KUKA KRL program: MyProgram_132().src

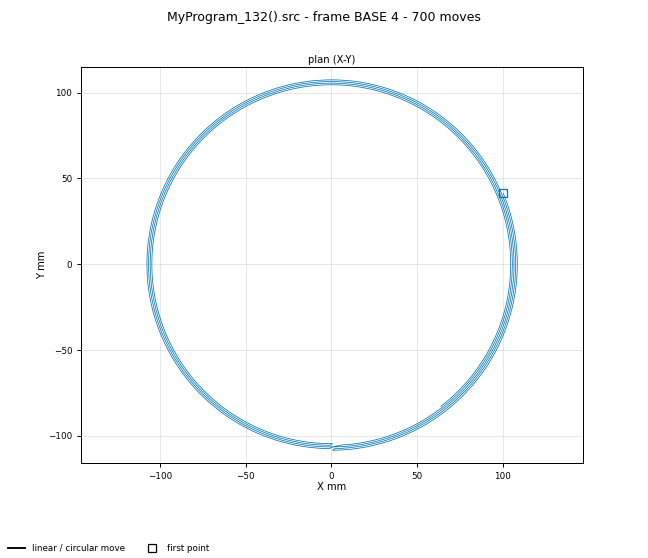
[picture p0: tool path of MyProgram_132().src in frame BASE 4, 700 of 700 moves have a stored position in this frame; points joined in program order, loops and branches not executed]
&ACCESS RVP
&REL 1
&PARAM TEMPLATE = C:\KRC\Roboter\Template\vorgabe
&PARAM EDITMASK = *
DEF MyProgram_132()
; ---- Setting reference (Base) ----
$BASE = BASE_DATA[4]

; --------------------------
; ---- Setting tool (TCP) ----
$TOOL = TOOL_DATA[3]
; --------------------------

$VEL.CP = VEL_APROX_PRINT
Startdeposition()
$VEL.CP = VEL_PRINT
LIN {X 100.2174,Y 41.413,Z 108,A 17.7358,B 24.9349,C -1.8633,E1 25.148,E2 427.9608} C_DIS
LIN {X 101.3618,Y 38.5229,Z 108,A 15.9205,B 24.9358,C -1.851,E1 25.1499,E2 429.795} C_DIS
LIN {X 102.6598,Y 34.9179,Z 108,A 13.9537,B 24.936,C -1.8475,E1 25.1517,E2 431.7591} C_DIS
LIN {X 103.7872,Y 31.4133,Z 108,A 11.2694,B 24.9386,C -1.8096,E1 25.154,E2 434.5174} C_DIS
LIN {X 105.0738,Y 26.7911,Z 108,A 10.0153,B 24.9353,C -1.8575,E1 25.1548,E2 435.6515} C_DIS
LIN {X 105.9493,Y 23.0863,Z 108,A 7.5492,B 24.9371,C -1.8313,E1 25.1564,E2 438.165} C_DIS
LIN {X 107.0471,Y 17.303,Z 108,A 4.2698,B 24.9383,C -1.8141,E1 25.158,E2 441.4657} C_DIS
LIN {X 107.5578,Y 13.7682,Z 108,A 2.4721,B 24.9385,C -1.812,E1 25.1587,E2 443.2578} C_DIS
LIN {X 107.9825,Y 9.8995,Z 108,A 0.4351,B 24.9388,C -1.8063,E1 25.1592,E2 445.2963} C_DIS
LIN {X 108.2207,Y 6.8359,Z 108,A -0.995,B 24.9386,C -1.8095,E1 25.1595,E2 446.7103} C_DIS
LIN {X 108.3454,Y 4.4221,Z 108,A -2.2285,B 24.9388,C -1.8073,E1 25.1597,E2 447.9416} C_DIS
LIN {X 108.4297,Y 1.2587,Z 108,A -4.0953,B 24.9397,C -1.7933,E1 25.1597,E2 449.8302} C_DIS
LIN {X 108.4149,Y -2.108,Z 108,A -5.7459,B 24.9397,C -1.7933,E1 25.1597,E2 451.4713} C_DIS
LIN {X 108.3146,Y -5.134,Z 108,A -7.3363,B 24.9401,C -1.7884,E1 25.1596,E2 453.0635} C_DIS
LIN {X 108.0913,Y -8.6313,Z 108,A -9.24,B 24.9406,C -1.7801,E1 25.1592,E2 454.9754} C_DIS
LIN {X 107.821,Y -11.5289,Z 108,A -10.7868,B 24.941,C -1.7747,E1 25.1587,E2 456.5258} C_DIS
LIN {X 107.3524,Y -15.287,Z 108,A -12.7437,B 24.9413,C -1.7702,E1 25.158,E2 458.4818} C_DIS
LIN {X 106.9242,Y -18.0404,Z 108,A -14.3021,B 24.9418,C -1.7617,E1 25.1573,E2 460.0513} C_DIS
LIN {X 106.2009,Y -21.8998,Z 108,A -16.2242,B 24.9418,C -1.7617,E1 25.1563,E2 461.9621} C_DIS
LIN {X 105.4391,Y -25.3175,Z 108,A -18.1427,B 24.9424,C -1.7527,E1 25.1551,E2 463.8905} C_DIS
LIN {X 104.5654,Y -28.714,Z 108,A -19.8437,B 24.9424,C -1.7535,E1 25.1539,E2 465.5799} C_DIS
LIN {X 103.5484,Y -32.1864,Z 108,A -21.8375,B 24.943,C -1.7439,E1 25.1523,E2 467.5851} C_DIS
LIN {X 102.2005,Y -36.2409,Z 108,A -24.0874,B 24.9434,C -1.7371,E1 25.1502,E2 469.8383} C_DIS
LIN {X 101.2136,Y -38.9144,Z 108,A -25.7145,B 24.9441,C -1.7271,E1 25.1486,E2 471.4799} C_DIS
LIN {X 99.6341,Y -42.7972,Z 108,A -27.9037,B 24.9445,C -1.7214,E1 25.1462,E2 473.6705} C_DIS
LIN {X 97.9263,Y -46.571,Z 108,A -29.7606,B 24.944,C -1.7293,E1 25.1441,E2 475.4988} C_DIS
LIN {X 96.5001,Y -49.4566,Z 108,A -31.55,B 24.9445,C -1.7203,E1 25.1419,E2 477.2998} C_DIS
LIN {X 95.0328,Y -52.224,Z 108,A -33.2033,B 24.9449,C -1.7155,E1 25.1397,E2 478.9558} C_DIS
LIN {X 93.8125,Y -54.3839,Z 108,A -35.0766,B 24.9467,C -1.6872,E1 25.137,E2 480.8862} C_DIS
LIN {X 91.9194,Y -57.5243,Z 108,A -36.4571,B 24.9455,C -1.7058,E1 25.135,E2 482.2157} C_DIS
LIN {X 90.0598,Y -60.3962,Z 108,A -38.3961,B 24.9462,C -1.695,E1 25.132,E2 484.1706} C_DIS
LIN {X 88.1742,Y -63.1155,Z 108,A -40.3404,B 24.947,C -1.6816,E1 25.1288,E2 486.137} C_DIS
LIN {X 85.536,Y -66.6493,Z 108,A -42.4786,B 24.9469,C -1.6836,E1 25.1252,E2 488.2604} C_DIS
LIN {X 83.0321,Y -69.7439,Z 108,A -44.5732,B 24.9472,C -1.6784,E1 25.1215,E2 490.3575} C_DIS
LIN {X 80.3621,Y -72.805,Z 108,A -46.6647,B 24.9474,C -1.6752,E1 25.1176,E2 492.4472} C_DIS
LIN {X 78.4248,Y -74.8861,Z 108,A -48.6384,B 24.9489,C -1.6512,E1 25.1137,E2 494.469} C_DIS
LIN {X 75.6077,Y -77.7299,Z 108,A -50.0261,B 24.9473,C -1.6773,E1 25.1111,E2 495.7892} C_DIS
LIN {X 72.5545,Y -80.5864,Z 108,A -52.2321,B 24.9476,C -1.6722,E1 25.1066,E2 497.9982} C_DIS
LIN {X 70.9665,Y -81.9891,Z 108,A -53.4015,B 24.9479,C -1.6675,E1 25.1041,E2 499.1742} C_DIS
LIN {X 66.5838,Y -85.5866,Z 108,A -56.3229,B 24.9481,C -1.664,E1 25.0978,E2 502.0928} C_DIS
LIN {X 64.1554,Y -87.4204,Z 108,A -58.1267,B 24.9488,C -1.6522,E1 25.0937,E2 503.918} C_DIS
LIN {X 61.403,Y -89.377,Z 108,A -60.0545,B 24.9495,C -1.6424,E1 25.0892,E2 505.8623} C_DIS
LIN {X 58.1749,Y -91.5103,Z 108,A -61.8183,B 24.949,C -1.6504,E1 25.0852,E2 507.6014} C_DIS
LIN {X 55.8874,Y -92.9251,Z 108,A -63.3876,B 24.9495,C -1.6414,E1 25.0814,E2 509.1871} C_DIS
LIN {X 52.8049,Y -94.7094,Z 108,A -65.1841,B 24.9495,C -1.6417,E1 25.077,E2 510.9776} C_DIS
LIN {X 48.1333,Y -97.1669,Z 108,A -67.9347,B 24.9497,C -1.6386,E1 25.0702,E2 513.7279} C_DIS
LIN {X 44.9286,Y -98.6905,Z 108,A -69.6324,B 24.9494,C -1.6431,E1 25.066,E2 515.4106} C_DIS
LIN {X 42.9037,Y -99.5877,Z 108,A -71.1287,B 24.9504,C -1.6276,E1 25.0621,E2 516.94} C_DIS
LIN {X 39.0287,Y -101.1702,Z 108,A -73.1237,B 24.95,C -1.6335,E1 25.0569,E2 518.9164} C_DIS
LIN {X 36.0035,Y -102.2838,Z 108,A -74.9642,B 24.9505,C -1.6256,E1 25.0521,E2 520.7719} C_DIS
LIN {X 32.966,Y -103.3037,Z 108,A -76.5757,B 24.9505,C -1.6269,E1 25.0478,E2 522.3772} C_DIS
LIN {X 29.4881,Y -104.3488,Z 108,A -78.4878,B 24.9505,C -1.625,E1 25.0427,E2 524.2906} C_DIS
LIN {X 24.9348,Y -105.5309,Z 108,A -81.0794,B 24.9509,C -1.6181,E1 25.0356,E2 526.8947} C_DIS
LIN {X 21.2833,Y -106.3275,Z 108,A -83.0284,B 24.9509,C -1.6174,E1 25.0303,E2 528.8429} C_DIS
LIN {X 17.7586,Y -106.9713,Z 108,A -84.8153,B 24.9509,C -1.6203,E1 25.0254,E2 530.6209} C_DIS
LIN {X 14.186,Y -107.5037,Z 108,A -86.8377,B 24.9512,C -1.6143,E1 25.0198,E2 532.6558} C_DIS
LIN {X 11.4639,Y -107.8278,Z 108,A -88.2968,B 24.9512,C -1.613,E1 25.0157,E2 534.1169} C_DIS
LIN {X 7.3656,Y -108.1849,Z 108,A -90.3919,B 24.9512,C -1.6152,E1 25.0099,E2 536.2058} C_DIS
LIN {X 3.338,Y -108.3839,Z 108,A -92.4794,B 24.9511,C -1.6162,E1 25.0041,E2 538.2903} C_DIS
LIN {X 0.7534,Y -108.4284,Z 108,A -93.489,B 24.9502,C -1.6305,E1 25.0014,E2 539.2659} C_DIS
Enddeposition()
LIN {X 0.7534,Y -108.4284,Z 108,A -93.489,B 24.9502,C -1.6305,E1 25.0014,E2 539.2659} C_DIS
Startdeposition()
$VEL.CP = VEL_PRINT
LIN {X 2.1755,Y -107.4555,Z 108,A -92.3471,B 24.9482,C -1.6631,E1 25.0048,E2 538.0468} C_DIS
LIN {X 5.6088,Y -107.3314,Z 108,A -90.697,B 24.9486,C -1.6563,E1 25.0093,E2 536.4133} C_DIS
LIN {X 10.474,Y -106.9674,Z 108,A -87.885,B 24.948,C -1.6663,E1 25.0172,E2 533.5792} C_DIS
LIN {X 16.3696,Y -106.2234,Z 108,A -84.7358,B 24.9479,C -1.6676,E1 25.0259,E2 530.4295} C_DIS
LIN {X 19.8404,Y -105.6313,Z 108,A -82.7772,B 24.9476,C -1.6725,E1 25.0313,E2 528.4615} C_DIS
LIN {X 27.3928,Y -103.93,Z 108,A -78.6876,B 24.9474,C -1.6748,E1 25.0425,E2 524.3721} C_DIS
LIN {X 30.6219,Y -103.0227,Z 108,A -76.8785,B 24.9473,C -1.6778,E1 25.0473,E2 522.5591} C_DIS
LIN {X 34.9072,Y -101.6524,Z 108,A -74.5529,B 24.9473,C -1.6776,E1 25.0535,E2 520.2383} C_DIS
LIN {X 38.1968,Y -100.4609,Z 108,A -72.6586,B 24.947,C -1.6814,E1 25.0584,E2 518.3392} C_DIS
LIN {X 42.2535,Y -98.8247,Z 108,A -70.4995,B 24.9473,C -1.6774,E1 25.064,E2 516.1944} C_DIS
LIN {X 46.3348,Y -96.9769,Z 108,A -67.994,B 24.9467,C -1.6861,E1 25.0704,E2 513.6746} C_DIS
LIN {X 48.6059,Y -95.8591,Z 108,A -66.4786,B 24.9461,C -1.6955,E1 25.0742,E2 512.1413} C_DIS
LIN {X 55.1038,Y -92.2777,Z 108,A -62.6335,B 24.946,C -1.6978,E1 25.0835,E2 508.3022} C_DIS
LIN {X 60.9574,Y -88.52,Z 108,A -58.7726,B 24.9451,C -1.7116,E1 25.0926,E2 504.4213} C_DIS
LIN {X 64.2874,Y -86.1314,Z 108,A -56.7712,B 24.9453,C -1.7083,E1 25.097,E2 502.4349} C_DIS
LIN {X 68.3346,Y -82.9568,Z 108,A -53.9272,B 24.9446,C -1.7188,E1 25.1033,E2 499.5769} C_DIS
LIN {X 71.9828,Y -79.8123,Z 108,A -51.6167,B 24.945,C -1.7135,E1 25.1081,E2 497.2878} C_DIS
LIN {X 74.8163,Y -77.1622,Z 108,A -49.2313,B 24.9438,C -1.7323,E1 25.1129,E2 494.868} C_DIS
LIN {X 78.486,Y -73.4262,Z 108,A -46.4053,B 24.9432,C -1.7408,E1 25.1184,E2 492.0343} C_DIS
LIN {X 81.4797,Y -70.0907,Z 108,A -44.263,B 24.9435,C -1.7361,E1 25.1223,E2 489.9125} C_DIS
LIN {X 83.9877,Y -67.0649,Z 108,A -41.9527,B 24.9425,C -1.7511,E1 25.1264,E2 487.5775} C_DIS
LIN {X 88.9292,Y -60.3571,Z 108,A -38.0875,B 24.9434,C -1.7381,E1 25.1327,E2 483.7618} C_DIS
LIN {X 92.9254,Y -54.0049,Z 108,A -33.8256,B 24.9419,C -1.7609,E1 25.139,E2 479.4677} C_DIS
LIN {X 94.725,Y -50.7821,Z 108,A -31.9145,B 24.9417,C -1.7642,E1 25.1415,E2 477.5588} C_DIS
LIN {X 96.4995,Y -47.3225,Z 108,A -29.9065,B 24.9414,C -1.7676,E1 25.144,E2 475.5536} C_DIS
LIN {X 98.1165,Y -43.8706,Z 108,A -27.904,B 24.9411,C -1.7725,E1 25.1464,E2 473.5504} C_DIS
LIN {X 99.2988,Y -41.1284,Z 108,A -26.2607,B 24.9406,C -1.7796,E1 25.1482,E2 471.8993} C_DIS
LIN {X 100.7196,Y -37.5138,Z 108,A -23.6154,B 24.9385,C -1.8115,E1 25.1508,E2 469.1935} C_DIS
LIN {X 102.0856,Y -33.6188,Z 108,A -21.9749,B 24.9397,C -1.7936,E1 25.1523,E2 467.6046} C_DIS
LIN {X 102.8525,Y -31.1955,Z 108,A -20.449,B 24.9389,C -1.8054,E1 25.1535,E2 466.0594} C_DIS
LIN {X 104.205,Y -26.323,Z 108,A -17.9238,B 24.9389,C -1.8064,E1 25.1553,E2 463.5463} C_DIS
LIN {X 105.0191,Y -22.8553,Z 108,A -16.2176,B 24.9389,C -1.8041,E1 25.1564,E2 461.8556} C_DIS
LIN {X 106.0556,Y -17.4263,Z 108,A -13.2387,B 24.9383,C -1.815,E1 25.1579,E2 458.8684} C_DIS
LIN {X 106.7848,Y -12.1855,Z 108,A -10.3746,B 24.9375,C -1.826,E1 25.1589,E2 455.9953} C_DIS
LIN {X 107.1337,Y -8.5882,Z 108,A -8.504,B 24.9372,C -1.8298,E1 25.1594,E2 454.1267} C_DIS
LIN {X 107.3094,Y -6.0066,Z 108,A -6.7645,B 24.9358,C -1.8502,E1 25.1597,E2 452.3495} C_DIS
LIN {X 107.4778,Y -0.1201,Z 108,A -4.106,B 24.9366,C -1.8391,E1 25.1597,E2 449.7329} C_DIS
LIN {X 107.445,Y 2.7028,Z 108,A -2.608,B 24.9363,C -1.8436,E1 25.1597,E2 448.2331} C_DIS
LIN {X 107.2976,Y 6.2204,Z 108,A -0.7097,B 24.9358,C -1.8506,E1 25.1595,E2 446.3296} C_DIS
LIN {X 106.8276,Y 11.8152,Z 108,A 2.4628,B 24.9346,C -1.8681,E1 25.1586,E2 443.1348} C_DIS
LIN {X 105.8604,Y 18.5786,Z 108,A 6.0922,B 24.9338,C -1.879,E1 25.1571,E2 439.5009} C_DIS
LIN {X 104.7521,Y 24.05,Z 108,A 8.6705,B 24.9344,C -1.8709,E1 25.1556,E2 436.9568} C_DIS
LIN {X 104.1786,Y 26.4258,Z 108,A 10.9566,B 24.931,C -1.9181,E1 25.154,E2 434.5725} C_DIS
LIN {X 102.9034,Y 31.0242,Z 108,A 12.8371,B 24.9326,C -1.8966,E1 25.1526,E2 432.7534} C_DIS
LIN {X 101.7298,Y 34.6777,Z 108,A 14.6618,B 24.9328,C -1.8931,E1 25.151,E2 430.9473} C_DIS
LIN {X 100.7146,Y 37.5269,Z 108,A 16.3732,B 24.9322,C -1.9022,E1 25.1493,E2 429.224} C_DIS
LIN {X 99.3665,Y 40.9621,Z 108,A 18.168,B 24.9322,C -1.9005,E1 25.1475,E2 427.4432} C_DIS
LIN {X 97.582,Y 45.0471,Z 108,A 20.6231,B 24.9316,C -1.9107,E1 25.1447,E2 424.9774} C_DIS
LIN {X 95.3511,Y 49.5968,Z 108,A 23.4592,B 24.9306,C -1.9241,E1 25.1411,E2 422.1248} C_DIS
LIN {X 93.5604,Y 52.8976,Z 108,A 25.4853,B 24.9301,C -1.9306,E1 25.1384,E2 420.0939} C_DIS
LIN {X 91.7671,Y 55.9481,Z 108,A 27.1655,B 24.9304,C -1.9268,E1 25.136,E2 418.4314} C_DIS
LIN {X 90.294,Y 58.2962,Z 108,A 28.7524,B 24.9298,C -1.9353,E1 25.1336,E2 416.8322} C_DIS
LIN {X 87.0843,Y 62.9927,Z 108,A 31.782,B 24.9292,C -1.9429,E1 25.1287,E2 413.7998} C_DIS
LIN {X 84.7875,Y 66.0513,Z 108,A 34.0008,B 24.9283,C -1.9556,E1 25.1249,E2 411.5614} C_DIS
LIN {X 82.1809,Y 69.2676,Z 108,A 35.9569,B 24.9287,C -1.95,E1 25.1215,E2 409.6274} C_DIS
LIN {X 79.9786,Y 71.7971,Z 108,A 38.1128,B 24.9272,C -1.9699,E1 25.1174,E2 407.4341} C_DIS
LIN {X 77.7306,Y 74.2265,Z 108,A 39.5646,B 24.9279,C -1.9604,E1 25.1147,E2 406.0112} C_DIS
LIN {X 75.1913,Y 76.7976,Z 108,A 41.469,B 24.9277,C -1.9636,E1 25.1109,E2 404.1074} C_DIS
LIN {X 73.2451,Y 78.6562,Z 108,A 43.3,B 24.9262,C -1.9834,E1 25.1071,E2 402.2368} C_DIS
LIN {X 70.6337,Y 81.0078,Z 108,A 44.6842,B 24.9275,C -1.9663,E1 25.1043,E2 400.8986} C_DIS
LIN {X 67.8832,Y 83.3266,Z 108,A 46.3376,B 24.9281,C -1.9588,E1 25.1008,E2 399.2692} C_DIS
LIN {X 64.5086,Y 85.9652,Z 108,A 48.901,B 24.9269,C -1.9748,E1 25.0951,E2 396.6776} C_DIS
LIN {X 61.5492,Y 88.1087,Z 108,A 51.1388,B 24.9257,C -1.9903,E1 25.0899,E2 394.4108} C_DIS
LIN {X 57.5684,Y 90.7612,Z 108,A 53.4047,B 24.9263,C -1.9824,E1 25.0846,E2 392.1711} C_DIS
LIN {X 54.6985,Y 92.5173,Z 108,A 55.0245,B 24.9267,C -1.9778,E1 25.0808,E2 390.5671} C_DIS
LIN {X 50.772,Y 94.7305,Z 108,A 57.6285,B 24.9258,C -1.9895,E1 25.0744,E2 387.943} C_DIS
LIN {X 47.6223,Y 96.351,Z 108,A 59.5988,B 24.9253,C -1.9954,E1 25.0694,E2 385.9643} C_DIS
LIN {X 43.4947,Y 98.285,Z 108,A 61.9687,B 24.9253,C -1.9957,E1 25.0634,E2 383.5995} C_DIS
LIN {X 39.936,Y 99.7842,Z 108,A 63.8225,B 24.9258,C -1.9893,E1 25.0587,E2 381.765} C_DIS
LIN {X 35.8794,Y 101.3121,Z 108,A 65.9642,B 24.9262,C -1.9846,E1 25.0531,E2 379.6392} C_DIS
LIN {X 32.6895,Y 102.3863,Z 108,A 67.9603,B 24.9254,C -1.9943,E1 25.0478,E2 377.6238} C_DIS
LIN {X 29.8432,Y 103.2525,Z 108,A 69.4989,B 24.9254,C -1.9935,E1 25.0437,E2 376.0898} C_DIS
LIN {X 27.337,Y 103.9443,Z 108,A 71.0343,B 24.925,C -2.0005,E1 25.0395,E2 374.5402} C_DIS
LIN {X 24.124,Y 104.735,Z 108,A 72.7199,B 24.9251,C -1.9983,E1 25.0349,E2 372.8622} C_DIS
LIN {X 20.4136,Y 105.5209,Z 108,A 75.2445,B 24.9235,C -2.0198,E1 25.0279,E2 370.2898} C_DIS
LIN {X 16.7722,Y 106.1612,Z 108,A 76.9422,B 24.9243,C -2.0092,E1 25.0233,E2 368.6188} C_DIS
LIN {X 13.5336,Y 106.6222,Z 108,A 78.6697,B 24.9243,C -2.0089,E1 25.0185,E2 366.8933} C_DIS
LIN {X 8.9996,Y 107.1008,Z 108,A 80.7083,B 24.9255,C -1.9934,E1 25.013,E2 364.8929} C_DIS
LIN {X 4.4181,Y 107.3867,Z 108,A 83.3104,B 24.925,C -1.9996,E1 25.0057,E2 362.2772} C_DIS
LIN {X 1.2219,Y 107.4719,Z 108,A 85.5357,B 24.9235,C -2.0202,E1 24.9993,E2 360.003} C_DIS
LIN {X -2.3815,Y 107.4517,Z 108,A 87.2479,B 24.9241,C -2.0113,E1 24.9946,E2 358.3119} C_DIS
LIN {X -8.6943,Y 107.1252,Z 108,A 90.9767,B 24.9232,C -2.0243,E1 24.9841,E2 354.5508} C_DIS
LIN {X -12.9356,Y 106.6965,Z 108,A 92.7858,B 24.9247,C -2.0045,E1 24.9792,E2 352.7875} C_DIS
LIN {X -21.1225,Y 105.3825,Z 108,A 97.0042,B 24.9255,C -1.9932,E1 24.9677,E2 348.5919} C_DIS
LIN {X -23.806,Y 104.8084,Z 108,A 99.0321,B 24.9239,C -2.0142,E1 24.962,E2 346.5116} C_DIS
LIN {X -27.5052,Y 103.8997,Z 108,A 100.6617,B 24.9253,C -1.9963,E1 24.9577,E2 344.9221} C_DIS
LIN {X -31.2977,Y 102.8209,Z 108,A 102.5258,B 24.9261,C -1.9847,E1 24.9528,E2 343.0825} C_DIS
LIN {X -34.8101,Y 101.6851,Z 108,A 105.1163,B 24.9245,C -2.0066,E1 24.9458,E2 340.435} C_DIS
LIN {X -38.18,Y 100.4673,Z 108,A 106.5818,B 24.926,C -1.9868,E1 24.9421,E2 339.0136} C_DIS
LIN {X -41.7796,Y 99.0244,Z 108,A 109.5222,B 24.9236,C -2.0179,E1 24.9343,E2 335.9925} C_DIS
LIN {X -46.657,Y 96.8221,Z 108,A 111.4772,B 24.9266,C -1.9785,E1 24.9296,E2 334.1263} C_DIS
LIN {X -49.9614,Y 95.1591,Z 108,A 113.5112,B 24.9266,C -1.9776,E1 24.9245,E2 332.0888} C_DIS
LIN {X -53.2559,Y 93.3558,Z 108,A 115.4071,B 24.9272,C -1.97,E1 24.9199,E2 330.2054} C_DIS
LIN {X -55.8464,Y 91.8289,Z 108,A 117.095,B 24.9272,C -1.9704,E1 24.9159,E2 328.5117} C_DIS
LIN {X -58.9835,Y 89.8464,Z 108,A 118.9401,B 24.9279,C -1.9615,E1 24.9116,E2 326.6817} C_DIS
LIN {X -61.7414,Y 87.975,Z 108,A 121.4065,B 24.9262,C -1.9843,E1 24.9058,E2 324.1527} C_DIS
LIN {X -64.8457,Y 85.7108,Z 108,A 123.1237,B 24.9274,C -1.9673,E1 24.902,E2 322.4697} C_DIS
LIN {X -67.9403,Y 83.2803,Z 108,A 125.2611,B 24.9277,C -1.9642,E1 24.8974,E2 320.3316} C_DIS
LIN {X -71.5461,Y 80.2033,Z 108,A 127.7401,B 24.9282,C -1.9567,E1 24.8922,E2 317.8609} C_DIS
LIN {X -75.6079,Y 76.3861,Z 108,A 130.087,B 24.9304,C -1.9261,E1 24.8876,E2 315.5771} C_DIS
LIN {X -77.9442,Y 74.0017,Z 108,A 132.5306,B 24.929,C -1.9466,E1 24.8827,E2 313.0742} C_DIS
LIN {X -82.7601,Y 68.5723,Z 108,A 136.2051,B 24.9302,C -1.9293,E1 24.876,E2 309.4242} C_DIS
LIN {X -85.0114,Y 65.7608,Z 108,A 138.4369,B 24.9297,C -1.9359,E1 24.8721,E2 307.1662} C_DIS
LIN {X -87.8152,Y 61.9692,Z 108,A 140.8207,B 24.9306,C -1.9241,E1 24.8682,E2 304.799} C_DIS
LIN {X -90.1286,Y 58.5539,Z 108,A 142.8801,B 24.9314,C -1.9127,E1 24.8651,E2 302.7564} C_DIS
LIN {X -91.6849,Y 56.0835,Z 108,A 144.5754,B 24.9314,C -1.9135,E1 24.8626,E2 301.0506} C_DIS
LIN {X -93.6621,Y 52.7155,Z 108,A 146.571,B 24.932,C -1.9042,E1 24.8598,E2 299.0666} C_DIS
LIN {X -95.773,Y 48.7743,Z 108,A 149.0207,B 24.9324,C -1.8996,E1 24.8566,E2 296.6148} C_DIS
LIN {X -97.9592,Y 44.2197,Z 108,A 151.7733,B 24.9328,C -1.8937,E1 24.8534,E2 293.8614} C_DIS
LIN {X -99.3493,Y 41.0045,Z 108,A 153.7089,B 24.933,C -1.8905,E1 24.8513,E2 291.9226} C_DIS
LIN {X -100.9162,Y 36.9773,Z 108,A 155.6253,B 24.9345,C -1.8691,E1 24.8494,E2 290.0466} C_DIS
LIN {X -101.824,Y 34.3984,Z 108,A 157.342,B 24.9342,C -1.8741,E1 24.8478,E2 288.3082} C_DIS
LIN {X -102.9111,Y 30.9981,Z 108,A 159.312,B 24.9344,C -1.8706,E1 24.8462,E2 286.3353} C_DIS
LIN {X -103.9022,Y 27.4957,Z 108,A 161.383,B 24.9345,C -1.8692,E1 24.8447,E2 284.2554} C_DIS
LIN {X -104.8605,Y 23.5804,Z 108,A 163.4741,B 24.9351,C -1.8602,E1 24.8434,E2 282.1735} C_DIS
LIN {X -105.6701,Y 19.6313,Z 108,A 165.6739,B 24.9355,C -1.8552,E1 24.8422,E2 279.9727} C_DIS
LIN {X -106.708,Y 12.8412,Z 108,A 169.2529,B 24.9365,C -1.8403,E1 24.8408,E2 276.4079} C_DIS
LIN {X -107.0703,Y 9.359,Z 108,A 171.6427,B 24.9356,C -1.8537,E1 24.8402,E2 273.9718} C_DIS
LIN {X -107.335,Y 5.5429,Z 108,A 174.0238,B 24.9352,C -1.8599,E1 24.8398,E2 271.5615} C_DIS
LIN {X -107.4763,Y 0.3926,Z 108,A 175.5565,B 24.9389,C -1.8059,E1 24.8398,E2 270.1485} C_DIS
LIN {X -107.3137,Y -5.9289,Z 108,A 179.312,B 24.9387,C -1.8091,E1 24.8401,E2 266.3627} C_DIS
LIN {X -106.953,Y -10.6189,Z 108,A -178.0557,B 24.9389,C -1.8056,E1 24.8407,E2 263.7228} C_DIS
LIN {X -106.5754,Y -13.8949,Z 108,A -176.324,B 24.9393,C -1.7991,E1 24.8413,E2 261.9964} C_DIS
LIN {X -106.0516,Y -17.4503,Z 108,A -174.4404,B 24.9398,C -1.7918,E1 24.8421,E2 260.1189} C_DIS
LIN {X -105.3824,Y -21.1229,Z 108,A -172.4398,B 24.9402,C -1.786,E1 24.8432,E2 258.1205} C_DIS
LIN {X -104.7358,Y -24.1204,Z 108,A -170.769,B 24.9405,C -1.7823,E1 24.8442,E2 256.4487} C_DIS
LIN {X -103.798,Y -27.8813,Z 108,A -168.6915,B 24.9409,C -1.7763,E1 24.8457,E2 254.3733} C_DIS
LIN {X -102.9809,Y -30.7629,Z 108,A -167.1851,B 24.9414,C -1.7681,E1 24.8468,E2 252.8778} C_DIS
LIN {X -102.1079,Y -33.5499,Z 108,A -164.6641,B 24.9393,C -1.7997,E1 24.8491,E2 250.267} C_DIS
LIN {X -100.3352,Y -38.5289,Z 108,A -162.8217,B 24.9423,C -1.7546,E1 24.8508,E2 248.5218} C_DIS
LIN {X -98.2716,Y -43.5254,Z 108,A -159.7024,B 24.9423,C -1.7551,E1 24.8543,E2 245.384} C_DIS
LIN {X -96.6399,Y -47.0361,Z 108,A -157.6341,B 24.9426,C -1.7494,E1 24.8567,E2 243.3179} C_DIS
LIN {X -95.3672,Y -49.5662,Z 108,A -155.2984,B 24.9408,C -1.7766,E1 24.8599,E2 240.9049} C_DIS
LIN {X -92.7569,Y -54.2931,Z 108,A -153.5049,B 24.9441,C -1.7276,E1 24.8622,E2 239.2189} C_DIS
LIN {X -89.761,Y -59.113,Z 108,A -150.2259,B 24.944,C -1.7292,E1 24.8671,E2 235.9194} C_DIS
LIN {X -87.4793,Y -62.44,Z 108,A -148.2882,B 24.9448,C -1.7157,E1 24.8702,E2 234.0043} C_DIS
LIN {X -83.589,Y -67.5594,Z 108,A -144.7842,B 24.9452,C -1.7102,E1 24.8762,E2 230.4968} C_DIS
LIN {X -79.7864,Y -72.0117,Z 108,A -141.4749,B 24.9452,C -1.7102,E1 24.8822,E2 227.1726} C_DIS
LIN {X -77.1798,Y -74.798,Z 108,A -139.5526,B 24.9457,C -1.7014,E1 24.8859,E2 225.2627} C_DIS
LIN {X -72.2789,Y -79.5451,Z 108,A -135.8192,B 24.946,C -1.6975,E1 24.8935,E2 221.5233} C_DIS
LIN {X -67.3665,Y -83.7454,Z 108,A -132.2733,B 24.9462,C -1.6948,E1 24.9011,E2 217.9702} C_DIS
LIN {X -64.0732,Y -86.2923,Z 108,A -129.4171,B 24.9448,C -1.7158,E1 24.9076,E2 215.0538} C_DIS
LIN {X -60.3412,Y -88.94,Z 108,A -127.7461,B 24.947,C -1.6817,E1 24.9113,E2 213.4583} C_DIS
LIN {X -57.4757,Y -90.8202,Z 108,A -125.3045,B 24.9457,C -1.7029,E1 24.9171,E2 210.9584} C_DIS
LIN {X -54.0919,Y -92.8754,Z 108,A -123.6667,B 24.947,C -1.6812,E1 24.921,E2 209.3672} C_DIS
LIN {X -51.0829,Y -94.5619,Z 108,A -122.0046,B 24.9476,C -1.6718,E1 24.925,E2 207.7227} C_DIS
LIN {X -46.3804,Y -96.955,Z 108,A -119.0653,B 24.9476,C -1.6733,E1 24.9324,E2 204.7722} C_DIS
LIN {X -43.1946,Y -98.4158,Z 108,A -117.4847,B 24.9484,C -1.6598,E1 24.9363,E2 203.2197} C_DIS
LIN {X -39.3684,Y -100.0075,Z 108,A -114.9932,B 24.9478,C -1.6687,E1 24.9428,E2 200.7014} C_DIS
LIN {X -36.0536,Y -101.251,Z 108,A -113.1182,B 24.948,C -1.6665,E1 24.9477,E2 198.8279} C_DIS
LIN {X -31.47,Y -102.7675,Z 108,A -110.1759,B 24.9472,C -1.6793,E1 24.9556,E2 195.85} C_DIS
LIN {X -26.8894,Y -104.0594,Z 108,A -108.0556,B 24.9483,C -1.661,E1 24.9613,E2 193.7699} C_DIS
LIN {X -22.2513,Y -105.1499,Z 108,A -104.6243,B 24.9461,C -1.696,E1 24.9709,E2 190.2514} C_DIS
LIN {X -17.3286,Y -106.0719,Z 108,A -103.2714,B 24.9495,C -1.6416,E1 24.9742,E2 189.0262} C_DIS
LIN {X -13.1143,Y -106.676,Z 108,A -100.4816,B 24.9482,C -1.6621,E1 24.9821,E2 186.1856} C_DIS
LIN {X -8.7919,Y -107.1174,Z 108,A -98.1619,B 24.9482,C -1.6621,E1 24.9885,E2 183.8647} C_DIS
LIN {X -5.1823,Y -107.3538,Z 108,A -96.2966,B 24.9484,C -1.6595,E1 24.9937,E2 182.0048} C_DIS
LIN {X -1.1203,Y -107.4725,Z 108,A -93.6789,B 24.9472,C -1.6785,E1 25.0011,E2 179.342} C_DIS
LIN {X -1.1203,Y -107.4725,Z 108,A -93.6789,B 24.9472,C -1.6785,E1 25.0011,E2 179.342} C_DIS
Enddeposition()
LIN {X 0.7272,Y -106.4961,Z 108,A -92.7543,B 24.9463,C -1.693,E1 25.0038,E2 178.3831} C_DIS
Startdeposition()
$VEL.CP = VEL_PRINT
LIN {X -4.3116,Y -106.4323,Z 108,A -96.3794,B 24.9487,C -1.655,E1 24.9935,E2 182.0984} C_DIS
LIN {X -7.0999,Y -106.2825,Z 108,A -98.7857,B 24.9509,C -1.6191,E1 24.9865,E2 184.5907} C_DIS
LIN {X -11.2956,Y -105.9189,Z 108,A -100.319,B 24.9491,C -1.6481,E1 24.9824,E2 186.0559} C_DIS
LIN {X -15.9001,Y -105.3266,Z 108,A -102.9673,B 24.9494,C -1.6427,E1 24.9751,E2 188.7192} C_DIS
LIN {X -21.4369,Y -104.34,Z 108,A -106.1824,B 24.9498,C -1.6363,E1 24.9662,E2 191.9528} C_DIS
LIN {X -25.6481,Y -103.3862,Z 108,A -108.3153,B 24.9493,C -1.6449,E1 24.9604,E2 194.0681} C_DIS
LIN {X -29.0121,Y -102.4922,Z 108,A -110.8506,B 24.9508,C -1.6205,E1 24.9535,E2 196.6656} C_DIS
LIN {X -33.393,Y -101.1517,Z 108,A -112.521,B 24.9488,C -1.653,E1 24.9492,E2 198.2617} C_DIS
LIN {X -37.5486,Y -99.682,Z 108,A -114.9002,B 24.9487,C -1.6548,E1 24.943,E2 200.6413} C_DIS
LIN {X -43.0282,Y -97.4433,Z 108,A -118.6151,B 24.9497,C -1.6377,E1 24.9333,E2 204.4055} C_DIS
LIN {X -46.0438,Y -96.0538,Z 108,A -120.2736,B 24.9493,C -1.6447,E1 24.9291,E2 206.0515} C_DIS
LIN {X -49.149,Y -94.5042,Z 108,A -121.9046,B 24.9486,C -1.656,E1 24.9251,E2 207.6601} C_DIS
LIN {X -52.1101,Y -92.9029,Z 108,A -123.6357,B 24.9483,C -1.6616,E1 24.9209,E2 209.383} C_DIS
LIN {X -57.6427,Y -89.5751,Z 108,A -126.8205,B 24.9473,C -1.6777,E1 24.9134,E2 212.5392} C_DIS
LIN {X -62.4869,Y -86.2673,Z 108,A -130.1987,B 24.9475,C -1.6743,E1 24.9056,E2 215.9369} C_DIS
LIN {X -65.0583,Y -84.3433,Z 108,A -132.0763,B 24.9476,C -1.6717,E1 24.9014,E2 217.8274} C_DIS
LIN {X -70.209,Y -80.1068,Z 108,A -135.392,B 24.9466,C -1.6887,E1 24.8943,E2 221.1153} C_DIS
LIN {X -72.456,Y -78.0795,Z 108,A -138.0866,B 24.9488,C -1.6523,E1 24.8886,E2 223.9076} C_DIS
LIN {X -75.9856,Y -74.6501,Z 108,A -139.8676,B 24.9465,C -1.69,E1 24.8852,E2 225.6064} C_DIS
LIN {X -78.2285,Y -72.2967,Z 108,A -142.2409,B 24.9477,C -1.6707,E1 24.8806,E2 228.036} C_DIS
LIN {X -80.7845,Y -69.4294,Z 108,A -143.7979,B 24.9462,C -1.6943,E1 24.8778,E2 229.544} C_DIS
LIN {X -82.8535,Y -66.9454,Z 108,A -146.3705,B 24.9479,C -1.6677,E1 24.8732,E2 232.1917} C_DIS
LIN {X -85.9336,Y -62.9427,Z 108,A -148.1387,B 24.9453,C -1.7092,E1 24.8704,E2 233.8697} C_DIS
LIN {X -87.7352,Y -60.4079,Z 108,A -150.0292,B 24.9455,C -1.7054,E1 24.8673,E2 235.7786} C_DIS
LIN {X -91.1196,Y -55.169,Z 108,A -153.1131,B 24.9443,C -1.7241,E1 24.8628,E2 238.8335} C_DIS
LIN {X -92.3964,Y -53.0027,Z 108,A -155.3315,B 24.9461,C -1.6961,E1 24.8596,E2 241.1301} C_DIS
LIN {X -94.4877,Y -49.1804,Z 108,A -156.9496,B 24.944,C -1.7289,E1 24.8575,E2 242.6786} C_DIS
LIN {X -95.9186,Y -46.3252,Z 108,A -158.8255,B 24.944,C -1.728,E1 24.8552,E2 244.5668} C_DIS
LIN {X -97.3925,Y -43.1446,Z 108,A -161.1762,B 24.9448,C -1.7165,E1 24.8525,E2 246.9579} C_DIS
LIN {X -98.8241,Y -39.7536,Z 108,A -162.5675,B 24.943,C -1.7436,E1 24.8511,E2 248.2923} C_DIS
LIN {X -100.1371,Y -36.3173,Z 108,A -165.0504,B 24.9438,C -1.7312,E1 24.8486,E2 250.8189} C_DIS
LIN {X -101.2248,Y -33.1671,Z 108,A -166.2344,B 24.942,C -1.7586,E1 24.8476,E2 251.9443} C_DIS
LIN {X -102.122,Y -30.2896,Z 108,A -167.906,B 24.9418,C -1.7617,E1 24.8462,E2 253.6181} C_DIS
LIN {X -102.9741,Y -27.2578,Z 108,A -169.7502,B 24.9418,C -1.7614,E1 24.8449,E2 255.4738} C_DIS
LIN {X -103.8011,Y -23.9102,Z 108,A -171.6401,B 24.9416,C -1.7659,E1 24.8436,E2 257.364} C_DIS
LIN {X -104.5573,Y -20.3515,Z 108,A -173.649,B 24.9413,C -1.7701,E1 24.8425,E2 259.3747} C_DIS
LIN {X -105.1799,Y -16.8493,Z 108,A -175.6512,B 24.9411,C -1.7729,E1 24.8416,E2 261.3822} C_DIS
LIN {X -105.7204,Y -13.0375,Z 108,A -177.7279,B 24.9407,C -1.7792,E1 24.8408,E2 263.456} C_DIS
LIN {X -106.119,Y -9.2426,Z 108,A 179.9317,B 24.9409,C -1.7755,E1 24.8402,E2 265.8195} C_DIS
LIN {X -106.3685,Y -5.671,Z 108,A 177.6909,B 24.9413,C -1.7705,E1 24.8399,E2 268.0857} C_DIS
LIN {X -106.5137,Y -1.2552,Z 108,A 176.0369,B 24.939,C -1.8039,E1 24.8399,E2 269.6699} C_DIS
LIN {X -106.386,Y 5.3538,Z 108,A 172.023,B 24.9393,C -1.799,E1 24.8401,E2 273.7197} C_DIS
LIN {X -106.0109,Y 10.4139,Z 108,A 169.5218,B 24.9382,C -1.816,E1 24.8407,E2 276.1954} C_DIS
LIN {X -105.6089,Y 13.8984,Z 108,A 167.2429,B 24.9387,C -1.8081,E1 24.8415,E2 278.5068} C_DIS
LIN {X -105.0743,Y 17.4858,Z 108,A 166.1392,B 24.9362,C -1.8448,E1 24.842,E2 279.5296} C_DIS
LIN {X -104.4712,Y 20.7975,Z 108,A 164.041,B 24.9365,C -1.8402,E1 24.8431,E2 281.6512} C_DIS
LIN {X -103.6763,Y 24.4506,Z 108,A 161.9943,B 24.9362,C -1.8453,E1 24.8443,E2 283.6976} C_DIS
LIN {X -102.7213,Y 28.1938,Z 108,A 159.7611,B 24.9361,C -1.8463,E1 24.8459,E2 285.9414} C_DIS
LIN {X -101.6152,Y 31.9515,Z 108,A 157.612,B 24.9357,C -1.8515,E1 24.8476,E2 288.0906} C_DIS
LIN {X -100.3358,Y 35.7682,Z 108,A 155.3219,B 24.9356,C -1.8537,E1 24.8497,E2 290.3883} C_DIS
LIN {X -99.169,Y 38.883,Z 108,A 153.7084,B 24.9348,C -1.8656,E1 24.8514,E2 291.9827} C_DIS
LIN {X -97.7559,Y 42.3111,Z 108,A 151.1119,B 24.9358,C -1.8501,E1 24.8543,E2 294.6305} C_DIS
LIN {X -96.0617,Y 46.0274,Z 108,A 149.5551,B 24.9338,C -1.8797,E1 24.856,E2 296.1252} C_DIS
LIN {X -93.3219,Y 51.3597,Z 108,A 146.1085,B 24.9337,C -1.8811,E1 24.8605,E2 299.5867} C_DIS
LIN {X -91.5076,Y 54.5241,Z 108,A 144.236,B 24.933,C -1.8901,E1 24.8632,E2 301.4475} C_DIS
LIN {X -89.6996,Y 57.4487,Z 108,A 142.4816,B 24.9324,C -1.8988,E1 24.8657,E2 303.1901} C_DIS
LIN {X -88.0815,Y 59.9004,Z 108,A 140.8677,B 24.9322,C -1.902,E1 24.8683,E2 304.8045} C_DIS
LIN {X -86.0948,Y 62.7225,Z 108,A 138.533,B 24.9331,C -1.8897,E1 24.8721,E2 307.1797} C_DIS
LIN {X -83.9973,Y 65.5068,Z 108,A 137.2238,B 24.9312,C -1.9152,E1 24.8743,E2 308.4343} C_DIS
LIN {X -81.6795,Y 68.3737,Z 108,A 134.5813,B 24.9326,C -1.8965,E1 24.8791,E2 311.1336} C_DIS
LIN {X -79.2801,Y 71.141,Z 108,A 132.4949,B 24.9326,C -1.8973,E1 24.883,E2 313.2274} C_DIS
LIN {X -76.4494,Y 74.1754,Z 108,A 130.9747,B 24.9303,C -1.9287,E1 24.8858,E2 314.6794} C_DIS
LIN {X -74.3416,Y 76.2892,Z 108,A 128.6212,B 24.9319,C -1.9053,E1 24.8906,E2 317.0986} C_DIS
LIN {X -71.3227,Y 79.1174,Z 108,A 126.5413,B 24.9312,C -1.9157,E1 24.8949,E2 319.162} C_DIS
LIN {X -68.5853,Y 81.5036,Z 108,A 125.1365,B 24.9294,C -1.9402,E1 24.8978,E2 320.514} C_DIS
LIN {X -66.5123,Y 83.2035,Z 108,A 123.5161,B 24.9297,C -1.9368,E1 24.9013,E2 322.1487} C_DIS
LIN {X -60.3606,Y 87.7681,Z 108,A 119.4004,B 24.929,C -1.9454,E1 24.9106,E2 326.2582} C_DIS
LIN {X -57.2589,Y 89.8215,Z 108,A 117.4223,B 24.9287,C -1.9501,E1 24.9152,E2 328.2315} C_DIS
LIN {X -54.3385,Y 91.6173,Z 108,A 115.6099,B 24.9284,C -1.9547,E1 24.9195,E2 330.0386} C_DIS
LIN {X -51.6054,Y 93.1847,Z 108,A 113.7725,B 24.9285,C -1.9524,E1 24.924,E2 331.8869} C_DIS
LIN {X -48.49,Y 94.8424,Z 108,A 112.0454,B 24.9278,C -1.9619,E1 24.9282,E2 333.596} C_DIS
LIN {X -45.6351,Y 96.2489,Z 108,A 109.5284,B 24.9298,C -1.9346,E1 24.9348,E2 336.1843} C_DIS
LIN {X -41.3765,Y 98.1547,Z 108,A 107.7991,B 24.9274,C -1.9674,E1 24.939,E2 337.8398} C_DIS
LIN {X -36.6819,Y 100.0042,Z 108,A 104.6609,B 24.9283,C -1.9551,E1 24.9473,E2 341.0139} C_DIS
LIN {X -33.6557,Y 101.0634,Z 108,A 103.382,B 24.9269,C -1.974,E1 24.9506,E2 342.2502} C_DIS
LIN {X -31.5278,Y 101.7465,Z 108,A 102.0682,B 24.9272,C -1.9711,E1 24.9541,E2 343.5731} C_DIS
LIN {X -27.6306,Y 102.8734,Z 108,A 99.3295,B 24.9285,C -1.9524,E1 24.9616,E2 346.3607} C_DIS
LIN {X -23.7198,Y 103.8451,Z 108,A 97.7411,B 24.9268,C -1.9763,E1 24.9658,E2 347.8942} C_DIS
LIN {X -20.2474,Y 104.5773,Z 108,A 95.1553,B 24.9286,C -1.9521,E1 24.973,E2 350.5403} C_DIS
LIN {X -15.8978,Y 105.327,Z 108,A 93.7646,B 24.9256,C -1.9914,E1 24.9766,E2 351.8391} C_DIS
LIN {X -10.2729,Y 106.0239,Z 108,A 90.3518,B 24.9266,C -1.979,E1 24.9862,E2 355.2835} C_DIS
LIN {X -3.6308,Y 106.458,Z 108,A 86.721,B 24.9266,C -1.9784,E1 24.9963,E2 358.9168} C_DIS
LIN {X 1.8123,Y 106.504,Z 108,A 84.2187,B 24.9253,C -1.9957,E1 25.0032,E2 361.3783} C_DIS
LIN {X 7.8248,Y 106.2335,Z 108,A 79.9781,B 24.9282,C -1.9565,E1 25.0152,E2 365.7101} C_DIS
LIN {X 12.1004,Y 105.8302,Z 108,A 78.3877,B 24.9262,C -1.9843,E1 25.0195,E2 367.2335} C_DIS
LIN {X 15.1949,Y 105.4302,Z 108,A 75.7357,B 24.929,C -1.9457,E1 25.0271,E2 369.9745} C_DIS
LIN {X 20.5513,Y 104.5188,Z 108,A 74.2109,B 24.925,C -1.9997,E1 25.0309,E2 371.3699} C_DIS
LIN {X 24.4775,Y 103.67,Z 108,A 71.6628,B 24.9263,C -1.9831,E1 25.0379,E2 373.9539} C_DIS
LIN {X 28.2834,Y 102.6971,Z 108,A 69.3163,B 24.9271,C -1.9725,E1 25.0443,E2 376.3219} C_DIS
LIN {X 31.9112,Y 101.6277,Z 108,A 67.2559,B 24.9272,C -1.9699,E1 25.0498,E2 378.3847} C_DIS
LIN {X 35.392,Y 100.4678,Z 108,A 64.6318,B 24.9293,C -1.9423,E1 25.0569,E2 381.0689} C_DIS
LIN {X 40.1253,Y 98.6728,Z 108,A 63.1412,B 24.9258,C -1.9889,E1 25.0605,E2 382.4458} C_DIS
LIN {X 46.133,Y 96.011,Z 108,A 59.2709,B 24.9271,C -1.9712,E1 25.0704,E2 386.3485} C_DIS
LIN {X 49.0572,Y 94.5525,Z 108,A 57.3442,B 24.9278,C -1.962,E1 25.0752,E2 388.2916} C_DIS
LIN {X 54.7899,Y 91.35,Z 108,A 53.8845,B 24.928,C -1.9599,E1 25.0836,E2 391.7459} C_DIS
LIN {X 60.2501,Y 87.8447,Z 108,A 50.5644,B 24.9279,C -1.9613,E1 25.0914,E2 395.0519} C_DIS
LIN {X 63.8918,Y 85.2304,Z 108,A 47.1642,B 24.9311,C -1.9167,E1 25.0992,E2 398.5454} C_DIS
LIN {X 68.0921,Y 81.9136,Z 108,A 45.2351,B 24.9287,C -1.9501,E1 25.1032,E2 400.3881} C_DIS
LIN {X 73.116,Y 77.4625,Z 108,A 41.9279,B 24.9283,C -1.9554,E1 25.11,E2 403.6696} C_DIS
LIN {X 75.0709,Y 75.57,Z 108,A 40.0528,B 24.9298,C -1.9352,E1 25.1138,E2 405.5847} C_DIS
LIN {X 79.8925,Y 70.4543,Z 108,A 36.543,B 24.9296,C -1.938,E1 25.1205,E2 409.0723} C_DIS
LIN {X 83.6276,Y 65.9758,Z 108,A 33.317,B 24.9304,C -1.9269,E1 25.1262,E2 412.3098} C_DIS
LIN {X 85.5729,Y 63.4353,Z 108,A 31.4707,B 24.9311,C -1.9174,E1 25.1293,E2 414.1697} C_DIS
LIN {X 89.2657,Y 58.1237,Z 108,A 28.1902,B 24.9311,C -1.9168,E1 25.1345,E2 417.4354} C_DIS
LIN {X 90.7825,Y 55.7236,Z 108,A 26.5308,B 24.9318,C -1.9072,E1 25.137,E2 419.109} C_DIS
LIN {X 93.1598,Y 51.65,Z 108,A 24.1305,B 24.9318,C -1.9062,E1 25.1403,E2 421.4994} C_DIS
LIN {X 94.6245,Y 48.9164,Z 108,A 21.8978,B 24.9339,C -1.8777,E1 25.1432,E2 423.7874} C_DIS
LIN {X 96.2612,Y 45.6113,Z 108,A 20.2811,B 24.9332,C -1.8876,E1 25.1451,E2 425.3722} C_DIS
LIN {X 98.3625,Y 40.8835,Z 108,A 17.8849,B 24.9326,C -1.896,E1 25.1478,E2 427.7354} C_DIS
LIN {X 100.3162,Y 35.824,Z 108,A 14.8757,B 24.9335,C -1.8834,E1 25.1508,E2 430.7575} C_DIS
LIN {X 101.4936,Y 32.3364,Z 108,A 12.673,B 24.9346,C -1.868,E1 25.1527,E2 432.9842} C_DIS
LIN {X 103.3226,Y 25.9062,Z 108,A 9.3287,B 24.9346,C -1.8677,E1 25.1552,E2 436.31} C_DIS
LIN {X 103.9462,Y 23.2786,Z 108,A 7.138,B 24.9371,C -1.8317,E1 25.1566,E2 438.5728} C_DIS
LIN {X 104.7829,Y 19.1574,Z 108,A 5.3232,B 24.9363,C -1.8436,E1 25.1575,E2 440.3488} C_DIS
LIN {X 105.621,Y 13.8049,Z 108,A 2.6954,B 24.9361,C -1.8467,E1 25.1586,E2 442.954} C_DIS
LIN {X 106.2679,Y 7.3157,Z 108,A -0.5101,B 24.936,C -1.8484,E1 25.1594,E2 446.1364} C_DIS
LIN {X 106.4911,Y 2.5125,Z 108,A -3.2834,B 24.9371,C -1.8319,E1 25.1598,E2 448.932} C_DIS
LIN {X 106.4575,Y -3.6491,Z 108,A -7.5119,B 24.9405,C -1.7821,E1 25.1595,E2 453.2528} C_DIS
LIN {X 106.1755,Y -8.5519,Z 108,A -8.8979,B 24.9374,C -1.8274,E1 25.1593,E2 454.524} C_DIS
LIN {X 105.261,Y -16.3248,Z 108,A -13.0861,B 24.9383,C -1.8146,E1 25.1579,E2 458.7174} C_DIS
LIN {X 104.2927,Y -21.667,Z 108,A -16.3151,B 24.9398,C -1.7918,E1 25.1563,E2 461.9814} C_DIS
LIN {X 103.252,Y -26.1811,Z 108,A -19.5,B 24.9423,C -1.7542,E1 25.1541,E2 465.2367} C_DIS
LIN {X 102.1554,Y -30.1769,Z 108,A -21.0605,B 24.9409,C -1.7757,E1 25.153,E2 466.7375} C_DIS
LIN {X 101.1864,Y -33.2857,Z 108,A -23.6337,B 24.9436,C -1.735,E1 25.1507,E2 469.392} C_DIS
LIN {X 99.5678,Y -37.8501,Z 108,A -25.3687,B 24.9417,C -1.7641,E1 25.1491,E2 471.0489} C_DIS
LIN {X 98.6789,Y -40.1105,Z 108,A -26.7375,B 24.9421,C -1.7573,E1 25.1476,E2 472.426} C_DIS
LIN {X 97.2805,Y -43.394,Z 108,A -28.7074,B 24.9426,C -1.7493,E1 25.1454,E2 474.404} C_DIS
LIN {X 95.0797,Y -48.0257,Z 108,A -31.3177,B 24.9428,C -1.7473,E1 25.1422,E2 477.005} C_DIS
LIN {X 93.6292,Y -50.7932,Z 108,A -33.0444,B 24.9432,C -1.7404,E1 25.14,E2 478.7389} C_DIS
LIN {X 92.1187,Y -53.4859,Z 108,A -35.5767,B 24.9459,C -1.6985,E1 25.1363,E2 481.3569} C_DIS
LIN {X 89.3626,Y -57.9738,Z 108,A -37.2613,B 24.9433,C -1.7392,E1 25.1339,E2 482.9371} C_DIS
LIN {X 85.3126,Y -63.7824,Z 108,A -41.0129,B 24.9438,C -1.731,E1 25.1279,E2 486.6897} C_DIS
LIN {X 82.4145,Y -67.4871,Z 108,A -43.6676,B 24.9446,C -1.7189,E1 25.1233,E2 489.3605} C_DIS
LIN {X 77.8167,Y -72.7395,Z 108,A -48.0209,B 24.9469,C -1.6839,E1 25.1151,E2 493.7769} C_DIS
LIN {X 75.3216,Y -75.3202,Z 108,A -49.5204,B 24.946,C -1.6974,E1 25.1122,E2 495.2383} C_DIS
LIN {X 72.662,Y -77.8896,Z 108,A -51.6777,B 24.9468,C -1.6855,E1 25.1078,E2 497.4148} C_DIS
LIN {X 69.6272,Y -80.6149,Z 108,A -53.7598,B 24.9468,C -1.6851,E1 25.1034,E2 499.4895} C_DIS
LIN {X 66.4995,Y -83.2136,Z 108,A -55.8392,B 24.9468,C -1.6848,E1 25.099,E2 501.5618} C_DIS
LIN {X 63.8074,Y -85.2937,Z 108,A -58.2129,B 24.9485,C -1.6582,E1 25.0935,E2 503.9898} C_DIS
LIN {X 60.5118,Y -87.6631,Z 108,A -59.813,B 24.9472,C -1.678,E1 25.09,E2 505.5374} C_DIS
LIN {X 57.2617,Y -89.8197,Z 108,A -61.7316,B 24.947,C -1.6814,E1 25.0856,E2 507.4417} C_DIS
LIN {X 55.1217,Y -91.1483,Z 108,A -64.4197,B 24.9506,C -1.6237,E1 25.0788,E2 510.2578} C_DIS
LIN {X 49.4961,Y -94.3214,Z 108,A -66.7132,B 24.948,C -1.6663,E1 25.0734,E2 512.4442} C_DIS
LIN {X 46.1159,Y -96.0192,Z 108,A -69.6687,B 24.9505,C -1.6251,E1 25.0658,E2 515.4894} C_DIS
LIN {X 41.0994,Y -98.2715,Z 108,A -71.5551,B 24.9481,C -1.6647,E1 25.0612,E2 517.2777} C_DIS
LIN {X 38.2538,Y -99.4149,Z 108,A -73.4452,B 24.9488,C -1.6524,E1 25.0562,E2 519.1926} C_DIS
LIN {X 34.5665,Y -100.7563,Z 108,A -75.665,B 24.9493,C -1.6452,E1 25.0503,E2 521.425} C_DIS
LIN {X 30.2066,Y -102.1466,Z 108,A -77.8667,B 24.9488,C -1.653,E1 25.0445,E2 523.6043} C_DIS
LIN {X 27.1486,Y -103.0036,Z 108,A -80.0759,B 24.9502,C -1.6307,E1 25.0384,E2 525.8627} C_DIS
LIN {X 23.7035,Y -103.8489,Z 108,A -81.9527,B 24.9502,C -1.6302,E1 25.0333,E2 527.7382} C_DIS
LIN {X 20.2628,Y -104.5744,Z 108,A -83.3675,B 24.9491,C -1.6479,E1 25.0296,E2 529.1094} C_DIS
LIN {X 17.6081,Y -105.0539,Z 108,A -85.7791,B 24.9515,C -1.6081,E1 25.0227,E2 531.6127} C_DIS
LIN {X 12.1228,Y -105.8276,Z 108,A -87.2658,B 24.948,C -1.6663,E1 25.0189,E2 532.9603} C_DIS
LIN {X 5.9968,Y -106.3504,Z 108,A -90.9003,B 24.9489,C -1.6513,E1 25.0087,E2 536.6285} C_DIS
LIN {X 0.7272,Y -106.4961,Z 108,A -92.7488,B 24.9464,C -1.6907,E1 25.0039,E2 538.383} C_DIS
Enddeposition()
LIN {X 0.7272,Y -106.4961,Z 108,A -92.7488,B 24.9464,C -1.6907,E1 25.0039,E2 538.383} C_DIS
Startdeposition()
$VEL.CP = VEL_PRINT
LIN {X 5.6737,Y -105.4088,Z 108,A -90.5068,B 24.9464,C -1.6897,E1 25.0101,E2 536.1441} C_DIS
LIN {X 12.305,Y -104.8417,Z 108,A -87.0956,B 24.9469,C -1.6834,E1 25.0195,E2 532.7498} C_DIS
LIN {X 17.8886,Y -104.0357,Z 108,A -83.6955,B 24.9459,C -1.6993,E1 25.029,E2 529.3153} C_DIS
LIN {X 21.048,Y -103.4418,Z 108,A -81.004,B 24.9433,C -1.74,E1 25.0366,E2 526.5307} C_DIS
LIN {X 26.9045,Y -102.0772,Z 108,A -78.7161,B 24.9457,C -1.7027,E1 25.0426,E2 524.3345} C_DIS
LIN {X 30.4741,Y -101.068,Z 108,A -76.764,B 24.9457,C -1.7025,E1 25.0478,E2 522.3864} C_DIS
LIN {X 32.7322,Y -100.3586,Z 108,A -75.3655,B 24.9453,C -1.7088,E1 25.0515,E2 520.9756} C_DIS
LIN {X 36.8498,Y -98.9222,Z 108,A -73.0475,B 24.9453,C -1.7098,E1 25.0576,E2 518.6599} C_DIS
LIN {X 41.668,Y -96.9895,Z 108,A -69.6119,B 24.9433,C -1.7398,E1 25.0666,E2 515.1613} C_DIS
LIN {X 45.897,Y -95.0615,Z 108,A -67.8393,B 24.945,C -1.7124,E1 25.0709,E2 513.4582} C_DIS
LIN {X 49.2823,Y -93.3512,Z 108,A -65.0419,B 24.9428,C -1.747,E1 25.078,E2 510.5869} C_DIS
LIN {X 53.3783,Y -91.0719,Z 108,A -63.2076,B 24.9445,C -1.7216,E1 25.0823,E2 508.8182} C_DIS
LIN {X 56.3734,Y -89.2497,Z 108,A -61.2819,B 24.9442,C -1.7262,E1 25.0869,E2 506.8878} C_DIS
LIN {X 58.6599,Y -87.7645,Z 108,A -59.6525,B 24.9436,C -1.7354,E1 25.0907,E2 505.242} C_DIS
LIN {X 64.0995,Y -83.8726,Z 108,A -56.371,B 24.944,C -1.7282,E1 25.098,E2 501.989} C_DIS
LIN {X 68.244,Y -80.5359,Z 108,A -53.5128,B 24.9437,C -1.7334,E1 25.1042,E2 499.1295} C_DIS
LIN {X 70.8699,Y -78.237,Z 108,A -51.5158,B 24.9431,C -1.7421,E1 25.1084,E2 497.1198} C_DIS
LIN {X 73.7359,Y -75.5421,Z 108,A -49.1236,B 24.9421,C -1.7582,E1 25.1133,E2 494.6996} C_DIS
LIN {X 77.1474,Y -72.0528,Z 108,A -46.6184,B 24.9421,C -1.7587,E1 25.1181,E2 492.204} C_DIS
LIN {X 80.2613,Y -68.5663,Z 108,A -44.2781,B 24.9421,C -1.7568,E1 25.1224,E2 489.8786} C_DIS
LIN {X 83.2929,Y -64.8499,Z 108,A -41.3498,B 24.9408,C -1.7777,E1 25.1275,E2 486.9147} C_DIS
LIN {X 86.9489,Y -59.8607,Z 108,A -38.2006,B 24.9408,C -1.778,E1 25.1326,E2 483.7801} C_DIS
LIN {X 88.8947,Y -56.9291,Z 108,A -36.5428,B 24.9411,C -1.7726,E1 25.1351,E2 482.1433} C_DIS
LIN {X 91.4216,Y -52.7762,Z 108,A -33.7793,B 24.9402,C -1.7856,E1 25.1391,E2 479.3633} C_DIS
LIN {X 93.138,Y -49.6872,Z 108,A -31.7949,B 24.9397,C -1.7941,E1 25.1418,E2 477.3693} C_DIS
LIN {X 94.5386,Y -46.9644,Z 108,A -29.8275,B 24.9384,C -1.8123,E1 25.1443,E2 475.3694} C_DIS
LIN {X 95.9838,Y -43.9393,Z 108,A -28.3167,B 24.939,C -1.8044,E1 25.146,E2 473.8854} C_DIS
LIN {X 97.2924,Y -40.9558,Z 108,A -26.4427,B 24.9383,C -1.8145,E1 25.1481,E2 471.998} C_DIS
LIN {X 98.7846,Y -37.2132,Z 108,A -23.7853,B 24.9364,C -1.8417,E1 25.1508,E2 469.2912} C_DIS
LIN {X 100.2906,Y -32.9425,Z 108,A -22.0178,B 24.938,C -1.8194,E1 25.1523,E2 467.5863} C_DIS
LIN {X 101.4184,Y -29.2878,Z 108,A -19.1243,B 24.935,C -1.8615,E1 25.1546,E2 464.6099} C_DIS
LIN {X 102.7234,Y -24.319,Z 108,A -17.1167,B 24.9368,C -1.8364,E1 25.1559,E2 462.6733} C_DIS
LIN {X 103.4546,Y -20.9858,Z 108,A -14.7102,B 24.9347,C -1.8665,E1 25.1572,E2 460.2097} C_DIS
LIN {X 104.2386,Y -16.667,Z 108,A -13.1432,B 24.9366,C -1.8387,E1 25.1579,E2 458.7174} C_DIS
LIN {X 105.053,Y -10.3656,Z 108,A -9.5579,B 24.9354,C -1.8557,E1 25.1592,E2 455.1132} C_DIS
LIN {X 105.296,Y -7.4883,Z 108,A -7.6649,B 24.9341,C -1.875,E1 25.1595,E2 453.1861} C_DIS
LIN {X 105.5597,Y 0.5029,Z 108,A -3.9218,B 24.9349,C -1.8632,E1 25.1598,E2 449.493} C_DIS
LIN {X 105.3234,Y 7.0836,Z 108,A 0.7396,B 24.9308,C -1.9218,E1 25.1591,E2 444.721} C_DIS
LIN {X 104.8329,Y 12.3803,Z 108,A 2.6943,B 24.933,C -1.8905,E1 25.1585,E2 442.8517} C_DIS
LIN {X 104.3688,Y 15.8253,Z 108,A 5.0848,B 24.931,C -1.9183,E1 25.1575,E2 440.4099} C_DIS
LIN {X 103.7439,Y 19.5089,Z 108,A 6.9177,B 24.9312,C -1.9162,E1 25.1566,E2 438.5927} C_DIS
LIN {X 102.7648,Y 24.1401,Z 108,A 9.234,B 24.9314,C -1.9133,E1 25.1552,E2 436.2967} C_DIS
LIN {X 102.085,Y 26.8733,Z 108,A 11.1035,B 24.93,C -1.9326,E1 25.1539,E2 434.3922} C_DIS
LIN {X 101.1836,Y 30.0846,Z 108,A 12.47,B 24.931,C -1.9191,E1 25.1528,E2 433.0655} C_DIS
LIN {X 100.0932,Y 33.5348,Z 108,A 14.402,B 24.9306,C -1.9236,E1 25.1511,E2 431.1338} C_DIS
LIN {X 99.2628,Y 35.9187,Z 108,A 16.1226,B 24.9292,C -1.9427,E1 25.1495,E2 429.3777} C_DIS
LIN {X 97.6256,Y 40.1568,Z 108,A 18.0637,B 24.9304,C -1.9274,E1 25.1475,E2 427.4834} C_DIS
LIN {X 95.0425,Y 45.9367,Z 108,A 21.8686,B 24.9285,C -1.9529,E1 25.1431,E2 423.6389} C_DIS
LIN {X 92.9645,Y 50.0093,Z 108,A 23.9575,B 24.9292,C -1.9431,E1 25.1404,E2 421.5844} C_DIS
LIN {X 91.9162,Y 51.912,Z 108,A 25.8712,B 24.9267,C -1.9776,E1 25.1377,E2 419.5991} C_DIS
LIN {X 89.8468,Y 55.4175,Z 108,A 27.599,B 24.9278,C -1.9629,E1 25.1352,E2 417.9149} C_DIS
LIN {X 85.9389,Y 61.3,Z 108,A 31.2821,B 24.9275,C -1.9663,E1 25.1295,E2 414.2419} C_DIS
LIN {X 83.7627,Y 64.2422,Z 108,A 33.2702,B 24.9271,C -1.9713,E1 25.1261,E2 412.2515} C_DIS
LIN {X 79.8021,Y 69.1014,Z 108,A 37.8923,B 24.9227,C -2.031,E1 25.1176,E2 407.5094} C_DIS
LIN {X 75.2853,Y 73.9959,Z 108,A 40.2501,B 24.9261,C -1.9857,E1 25.1132,E2 405.2689} C_DIS
LIN {X 72.9865,Y 76.2647,Z 108,A 42.9707,B 24.9227,C -2.03,E1 25.1075,E2 402.4547} C_DIS
LIN {X 68.8255,Y 80.0404,Z 108,A 45.0791,B 24.9253,C -1.9965,E1 25.1033,E2 400.4339} C_DIS
LIN {X 62.9467,Y 84.7421,Z 108,A 49.2026,B 24.9246,C -2.0055,E1 25.0942,E2 396.3043} C_DIS
LIN {X 59.7855,Y 87.0012,Z 108,A 51.106,B 24.925,C -2.0006,E1 25.0899,E2 394.4192} C_DIS
LIN {X 55.3002,Y 89.9188,Z 108,A 54.0525,B 24.9245,C -2.0069,E1 25.083,E2 391.4674} C_DIS
LIN {X 50.3256,Y 92.7929,Z 108,A 57.1828,B 24.9241,C -2.0118,E1 25.0754,E2 388.3348} C_DIS
LIN {X 47.094,Y 94.4743,Z 108,A 59.1901,B 24.9238,C -2.0156,E1 25.0704,E2 386.3241} C_DIS
LIN {X 44.8505,Y 95.5601,Z 108,A 61.2815,B 24.9214,C -2.0474,E1 25.0649,E2 384.1626} C_DIS
LIN {X 40.5327,Y 97.4707,Z 108,A 63.1851,B 24.9232,C -2.0232,E1 25.0601,E2 382.3209} C_DIS
LIN {X 34.9046,Y 99.6236,Z 108,A 66.1171,B 24.924,C -2.0126,E1 25.0526,E2 379.4202} C_DIS
LIN {X 32.7987,Y 100.3371,Z 108,A 67.6338,B 24.923,C -2.0261,E1 25.0485,E2 377.8744} C_DIS
LIN {X 29.2716,Y 101.423,Z 108,A 69.4896,B 24.9234,C -2.0216,E1 25.0435,E2 376.0325} C_DIS
LIN {X 26.0402,Y 102.2993,Z 108,A 71.4102,B 24.923,C -2.0269,E1 25.0383,E2 374.1023} C_DIS
LIN {X 22.5564,Y 103.1232,Z 108,A 73.2648,B 24.9232,C -2.0244,E1 25.0333,E2 372.2562} C_DIS
LIN {X 19.5188,Y 103.742,Z 108,A 75.5597,B 24.9212,C -2.0496,E1 25.0268,E2 369.9042} C_DIS
LIN {X 15.6148,Y 104.4013,Z 108,A 77.1426,B 24.9229,C -2.0276,E1 25.0226,E2 368.375} C_DIS
LIN {X 12.5747,Y 104.8101,Z 108,A 78.8437,B 24.9228,C -2.0294,E1 25.0179,E2 366.671} C_DIS
LIN {X 7.8436,Y 105.271,Z 108,A 81.3475,B 24.923,C -2.0266,E1 25.011,E2 364.1752} C_DIS
LIN {X 2.3808,Y 105.5354,Z 108,A 84.3581,B 24.9229,C -2.028,E1 25.0026,E2 361.1621} C_DIS
LIN {X -0.2686,Y 105.5616,Z 108,A 86.0814,B 24.922,C -2.039,E1 24.9977,E2 359.4128} C_DIS
LIN {X -4.9328,Y 105.4467,Z 108,A 88.779,B 24.9216,C -2.0446,E1 24.9901,E2 356.7013} C_DIS
LIN {X -8.3564,Y 105.23,Z 108,A 90.2063,B 24.923,C -2.0268,E1 24.9862,E2 355.3156} C_DIS
LIN {X -11.9523,Y 104.883,Z 108,A 92.5779,B 24.9218,C -2.0417,E1 24.9796,E2 352.9072} C_DIS
LIN {X -15.3217,Y 104.4445,Z 108,A 93.9106,B 24.9234,C -2.0207,E1 24.976,E2 351.6234} C_DIS
LIN {X -19.5089,Y 103.7439,Z 108,A 96.2115,B 24.9236,C -2.0188,E1 24.9697,E2 349.3247} C_DIS
LIN {X -22.7216,Y 103.0872,Z 108,A 98.2006,B 24.9231,C -2.0253,E1 24.9642,E2 347.3177} C_DIS
LIN {X -25.5643,Y 102.4204,Z 108,A 99.9652,B 24.9227,C -2.0307,E1 24.9594,E2 345.5378} C_DIS
LIN {X -30.253,Y 101.1336,Z 108,A 102.4348,B 24.9234,C -2.0214,E1 24.9528,E2 343.0865} C_DIS
LIN {X -37.5389,Y 98.6613,Z 108,A 106.5636,B 24.9239,C -2.0143,E1 24.942,E2 338.9665} C_DIS
LIN {X -40.7944,Y 97.3604,Z 108,A 108.3895,B 24.9243,C -2.0087,E1 24.9372,E2 337.1498} C_DIS
LIN {X -43.5536,Y 96.1578,Z 108,A 110.1418,B 24.9242,C -2.0107,E1 24.9328,E2 335.3884} C_DIS
LIN {X -47.7365,Y 94.1516,Z 108,A 112.581,B 24.9247,C -2.0037,E1 24.9267,E2 332.9595} C_DIS
LIN {X -50.9274,Y 92.466,Z 108,A 114.6955,B 24.9245,C -2.0062,E1 24.9214,E2 330.8331} C_DIS
LIN {X -54.3691,Y 90.4846,Z 108,A 116.796,B 24.925,C -2.0002,E1 24.9164,E2 328.7405} C_DIS
LIN {X -57.2972,Y 88.6585,Z 108,A 118.6884,B 24.9252,C -1.9974,E1 24.912,E2 326.8488} C_DIS
LIN {X -60.3389,Y 86.6165,Z 108,A 121.2001,B 24.924,C -2.0131,E1 24.9061,E2 324.2912} C_DIS
LIN {X -63.6547,Y 84.2103,Z 108,A 122.8777,B 24.9259,C -1.988,E1 24.9025,E2 322.6674} C_DIS
LIN {X -66.496,Y 81.9846,Z 108,A 124.8037,B 24.9263,C -1.9825,E1 24.8983,E2 320.7472} C_DIS
LIN {X -69.25,Y 79.6723,Z 108,A 126.9576,B 24.9261,C -1.9856,E1 24.8937,E2 318.5776} C_DIS
LIN {X -73.2697,Y 75.9917,Z 108,A 129.742,B 24.9271,C -1.9722,E1 24.888,E2 315.8137} C_DIS
LIN {X -75.8998,Y 73.3651,Z 108,A 131.747,B 24.9275,C -1.9668,E1 24.8841,E2 313.813} C_DIS
LIN {X -78.9081,Y 70.1202,Z 108,A 134.4298,B 24.9272,C -1.9711,E1 24.879,E2 311.1081} C_DIS
LIN {X -81.9188,Y 66.5772,Z 108,A 136.6709,B 24.9284,C -1.9541,E1 24.8751,E2 308.8971} C_DIS
LIN {X -83.9961,Y 63.9389,Z 108,A 138.77,B 24.928,C -1.9594,E1 24.8715,E2 306.7756} C_DIS
LIN {X -86.5756,Y 60.3977,Z 108,A 140.9322,B 24.9291,C -1.945,E1 24.868,E2 304.6372} C_DIS
LIN {X -88.5855,Y 57.411,Z 108,A 142.9761,B 24.9292,C -1.9427,E1 24.8648,E2 302.5882} C_DIS
LIN {X -90.1606,Y 54.9024,Z 108,A 144.607,B 24.9295,C -1.939,E1 24.8625,E2 300.9579} C_DIS
LIN {X -92.4345,Y 50.9839,Z 108,A 147.4652,B 24.929,C -1.9464,E1 24.8585,E2 298.0671} C_DIS
LIN {X -94.0414,Y 47.9522,Z 108,A 148.8119,B 24.9307,C -1.9221,E1 24.8568,E2 296.7712} C_DIS
LIN {X -95.1659,Y 45.6797,Z 108,A 150.8363,B 24.9293,C -1.9416,E1 24.8543,E2 294.6893} C_DIS
LIN {X -96.815,Y 42.0721,Z 108,A 152.4775,B 24.9312,C -1.9164,E1 24.8525,E2 293.0992} C_DIS
LIN {X -98.3314,Y 38.395,Z 108,A 154.6087,B 24.9317,C -1.9087,E1 24.8503,E2 290.9744} C_DIS
LIN {X -99.7493,Y 34.5463,Z 108,A 156.9506,B 24.9319,C -1.906,E1 24.8481,E2 288.6257} C_DIS
LIN {X -100.9933,Y 30.7221,Z 108,A 158.9461,B 24.9329,C -1.8923,E1 24.8465,E2 286.6514} C_DIS
LIN {X -101.6763,Y 28.3775,Z 108,A 160.4718,B 24.9327,C -1.8954,E1 24.8453,E2 285.1095} C_DIS
LIN {X -102.5738,Y 24.936,Z 108,A 162.3116,B 24.9333,C -1.886,E1 24.844,E2 283.2814} C_DIS
LIN {X -103.3956,Y 21.2731,Z 108,A 164.2144,B 24.9341,C -1.8746,E1 24.8429,E2 281.3945} C_DIS
LIN {X -104.0415,Y 17.8538,Z 108,A 166.6045,B 24.9333,C -1.8867,E1 24.8417,E2 278.9615} C_DIS
LIN {X -104.7664,Y 12.9441,Z 108,A 169.0737,B 24.9345,C -1.8698,E1 24.8408,E2 276.5178} C_DIS
LIN {X -105.1716,Y 9.083,Z 108,A 171.2388,B 24.9348,C -1.8651,E1 24.8402,E2 274.3509} C_DIS
LIN {X -105.4368,Y 5.1646,Z 108,A 173.5437,B 24.9348,C -1.8645,E1 24.8399,E2 272.0337} C_DIS
LIN {X -105.5584,Y 0.7433,Z 108,A 175.7008,B 24.936,C -1.8479,E1 24.8398,E2 269.9031} C_DIS
LIN {X -105.5348,Y -2.411,Z 108,A 177.7573,B 24.9355,C -1.8549,E1 24.8399,E2 267.8176} C_DIS
LIN {X -105.3773,Y -6.2436,Z 108,A 179.7397,B 24.9362,C -1.8445,E1 24.8402,E2 265.8479} C_DIS
LIN {X -105,Y -10.8725,Z 108,A -178.0307,B 24.9375,C -1.8259,E1 24.8408,E2 263.6494} C_DIS
LIN {X -104.6373,Y -13.9414,Z 108,A -176.2024,B 24.9375,C -1.826,E1 24.8414,E2 261.8098} C_DIS
LIN {X -104.077,Y -17.6417,Z 108,A -174.1676,B 24.9379,C -1.8198,E1 24.8423,E2 259.7779} C_DIS
LIN {X -103.4446,Y -21.0342,Z 108,A -172.4142,B 24.9386,C -1.8095,E1 24.8432,E2 258.0385} C_DIS
LIN {X -102.7208,Y -24.3303,Z 108,A -170.3542,B 24.9384,C -1.8122,E1 24.8445,E2 255.9602} C_DIS
LIN {X -101.7369,Y -28.1637,Z 108,A -168.2724,B 24.9391,C -1.8031,E1 24.846,E2 253.8877} C_DIS
LIN {X -100.6988,Y -31.6719,Z 108,A -166.4455,B 24.9399,C -1.7914,E1 24.8475,E2 252.0785} C_DIS
LIN {X -99.931,Y -34.0152,Z 108,A -164.6319,B 24.9389,C -1.8048,E1 24.8492,E2 250.2226} C_DIS
LIN {X -98.4018,Y -38.2156,Z 108,A -162.4927,B 24.9401,C -1.787,E1 24.8513,E2 248.1135} C_DIS
LIN {X -96.4197,Y -42.9723,Z 108,A -159.6914,B 24.9407,C -1.7791,E1 24.8543,E2 245.3155} C_DIS
LIN {X -94.9583,Y -46.1119,Z 108,A -157.8413,B 24.9411,C -1.7727,E1 24.8565,E2 243.4707} C_DIS
LIN {X -93.6081,Y -48.7945,Z 108,A -155.887,B 24.9406,C -1.7802,E1 24.8591,E2 241.4881} C_DIS
LIN {X -91.0875,Y -53.352,Z 108,A -153.298,B 24.9417,C -1.7637,E1 24.8626,E2 238.9248} C_DIS
LIN {X -89.4651,Y -56.0285,Z 108,A -151.2831,B 24.9412,C -1.771,E1 24.8656,E2 236.8823} C_DIS
LIN {X -87.7107,Y -58.7393,Z 108,A -149.9366,B 24.9425,C -1.7514,E1 24.8677,E2 235.5759} C_DIS
LIN {X -85.9389,Y -61.3,Z 108,A -148.2386,B 24.9428,C -1.7475,E1 24.8704,E2 233.8789} C_DIS
LIN {X -82.9212,Y -65.3245,Z 108,A -145.4641,B 24.9431,C -1.7424,E1 24.8751,E2 231.1031} C_DIS
LIN {X -80.8182,Y -67.9113,Z 108,A -143.5687,B 24.9431,C -1.7414,E1 24.8785,E2 229.2016} C_DIS
LIN {X -77.6798,Y -71.4771,Z 108,A -140.9706,B 24.9435,C -1.7363,E1 24.8833,E2 226.6038} C_DIS
LIN {X -75.8346,Y -73.4327,Z 108,A -139.5017,B 24.9437,C -1.7335,E1 24.8861,E2 225.1354} C_DIS
LIN {X -70.9484,Y -78.1654,Z 108,A -135.7674,B 24.9441,C -1.7274,E1 24.8937,E2 221.4002} C_DIS
LIN {X -68.2944,Y -80.4929,Z 108,A -133.4277,B 24.9433,C -1.7398,E1 24.8988,E2 219.0218} C_DIS
LIN {X -65.439,Y -82.8307,Z 108,A -131.9293,B 24.9448,C -1.7169,E1 24.9019,E2 217.5724} C_DIS
LIN {X -62.5654,Y -85.0225,Z 108,A -130.2434,B 24.9457,C -1.703,E1 24.9056,E2 215.9135} C_DIS
LIN {X -58.7791,Y -87.6838,Z 108,A -127.3889,B 24.9451,C -1.7118,E1 24.9123,E2 213.0283} C_DIS
LIN {X -55.9508,Y -89.5136,Z 108,A -125.2266,B 24.9444,C -1.7219,E1 24.9174,E2 210.8352} C_DIS
LIN {X -53.1411,Y -91.2119,Z 108,A -123.6786,B 24.9452,C -1.7102,E1 24.9211,E2 209.3103} C_DIS
LIN {X -49.695,Y -93.1339,Z 108,A -121.6163,B 24.9456,C -1.7043,E1 24.9261,E2 207.2563} C_DIS
LIN {X -47.1977,Y -94.4229,Z 108,A -119.5613,B 24.9444,C -1.723,E1 24.9314,E2 205.1514} C_DIS
LIN {X -43.6262,Y -96.1251,Z 108,A -118.0141,B 24.946,C -1.6972,E1 24.9352,E2 203.6617} C_DIS
LIN {X -40.8951,Y -97.318,Z 108,A -116.0492,B 24.9453,C -1.709,E1 24.9403,E2 201.6642} C_DIS
LIN {X -36.2997,Y -99.1238,Z 108,A -113.5998,B 24.946,C -1.6975,E1 24.9466,E2 199.237} C_DIS
LIN {X -32.6753,Y -100.377,Z 108,A -111.1333,B 24.9451,C -1.7109,E1 24.9533,E2 196.734} C_DIS
LIN {X -29.2711,Y -101.4231,Z 108,A -109.6201,B 24.9463,C -1.693,E1 24.9572,E2 195.2608} C_DIS
LIN {X -26.0802,Y -102.2891,Z 108,A -107.9239,B 24.9466,C -1.6881,E1 24.9618,E2 193.5738} C_DIS
LIN {X -22.9308,Y -103.0416,Z 108,A -105.9429,B 24.9461,C -1.696,E1 24.9672,E2 191.5713} C_DIS
LIN {X -18.0912,Y -104.0012,Z 108,A -103.2998,B 24.9462,C -1.6936,E1 24.9745,E2 188.9311} C_DIS
LIN {X -14.4402,Y -104.5698,Z 108,A -100.9355,B 24.9454,C -1.7075,E1 24.9811,E2 186.532} C_DIS
LIN {X -10.9394,Y -104.993,Z 108,A -99.6688,B 24.947,C -1.6814,E1 24.9845,E2 185.3264} C_DIS
LIN {X -6.6164,Y -105.355,Z 108,A -97.0942,B 24.9465,C -1.6901,E1 24.9917,E2 182.7301} C_DIS
LIN {X -0.6771,Y -105.5591,Z 108,A -94.0179,B 24.9468,C -1.6846,E1 25.0003,E2 179.6665} C_DIS
LIN {X -0.6771,Y -105.5591,Z 108,A -94.0179,B 24.9468,C -1.6846,E1 25.0003,E2 179.6665} C_DIS
Enddeposition()
LIN {X 0.6861,Y -104.5966,Z 108,A -93.2371,B 24.9456,C -1.7031,E1 25.0026,E2 178.842} C_DIS
Startdeposition()
$VEL.CP = VEL_PRINT
LIN {X -1.6768,Y -104.5901,Z 108,A -95.3483,B 24.9477,C -1.6704,E1 24.9964,E2 181.0305} C_DIS
LIN {X -5.155,Y -104.478,Z 108,A -97.6088,B 24.9486,C -1.6565,E1 24.99,E2 183.3247} C_DIS
LIN {X -9.7497,Y -104.148,Z 108,A -99.6893,B 24.9475,C -1.6737,E1 24.9844,E2 185.3652} C_DIS
LIN {X -13.1738,Y -103.7708,Z 108,A -101.657,B 24.9477,C -1.6709,E1 24.9789,E2 187.3409} C_DIS
LIN {X -16.7158,Y -103.2605,Z 108,A -103.6552,B 24.9477,C -1.6699,E1 24.9733,E2 189.3432} C_DIS
LIN {X -19.8002,Y -102.7122,Z 108,A -105.3451,B 24.9477,C -1.6715,E1 24.9687,E2 191.0309} C_DIS
LIN {X -22.9306,Y -102.0609,Z 108,A -107.1749,B 24.9477,C -1.6693,E1 24.9637,E2 192.8683} C_DIS
LIN {X -25.9695,Y -101.3284,Z 108,A -108.808,B 24.9475,C -1.6733,E1 24.9593,E2 194.4942} C_DIS
LIN {X -29.7698,Y -100.2777,Z 108,A -111.0694,B 24.9477,C -1.6709,E1 24.9532,E2 196.765} C_DIS
LIN {X -33.4331,Y -99.1165,Z 108,A -112.9138,B 24.947,C -1.6825,E1 24.9484,E2 198.5853} C_DIS
LIN {X -36.6681,Y -97.9666,Z 108,A -114.7351,B 24.9467,C -1.6864,E1 24.9436,E2 200.401} C_DIS
LIN {X -39.2536,Y -96.959,Z 108,A -116.2791,B 24.9467,C -1.6869,E1 24.9396,E2 201.9469} C_DIS
LIN {X -41.7941,Y -95.8911,Z 108,A -117.9748,B 24.947,C -1.6815,E1 24.9352,E2 203.6596} C_DIS
LIN {X -43.971,Y -94.9128,Z 108,A -119.4154,B 24.9472,C -1.6779,E1 24.9315,E2 205.1121} C_DIS
LIN {X -47.8628,Y -93.0112,Z 108,A -121.7515,B 24.947,C -1.6823,E1 24.9257,E2 207.4442} C_DIS
LIN {X -50.6902,Y -91.5012,Z 108,A -123.4748,B 24.9467,C -1.6858,E1 24.9215,E2 209.1639} C_DIS
LIN {X -52.8959,Y -90.2442,Z 108,A -124.952,B 24.9468,C -1.6846,E1 24.9179,E2 210.6484} C_DIS
LIN {X -56.5986,Y -87.9685,Z 108,A -127.1799,B 24.9462,C -1.6939,E1 24.9126,E2 212.8613} C_DIS
LIN {X -59.2448,Y -86.2103,Z 108,A -129.1123,B 24.9465,C -1.6896,E1 24.9081,E2 214.8104} C_DIS
LIN {X -62.4937,Y -83.8842,Z 108,A -131.1941,B 24.946,C -1.6973,E1 24.9035,E2 216.8811} C_DIS
LIN {X -64.7116,Y -82.1845,Z 108,A -132.8036,B 24.946,C -1.6972,E1 24.8999,E2 218.4968} C_DIS
LIN {X -67.7837,Y -79.6694,Z 108,A -134.8772,B 24.9455,C -1.705,E1 24.8955,E2 220.5597} C_DIS
LIN {X -70.6945,Y -77.0983,Z 108,A -137.8971,B 24.9473,C -1.6768,E1 24.8891,E2 223.6588} C_DIS
LIN {X -74.3962,Y -73.5327,Z 108,A -139.8265,B 24.9449,C -1.7149,E1 24.8854,E2 225.5058} C_DIS
LIN {X -77.9352,Y -69.7707,Z 108,A -142.6746,B 24.9445,C -1.7205,E1 24.88,E2 228.3531} C_DIS
LIN {X -80.2496,Y -67.0965,Z 108,A -144.6128,B 24.9442,C -1.7249,E1 24.8765,E2 230.2897} C_DIS
LIN {X -82.287,Y -64.5819,Z 108,A -146.3333,B 24.9438,C -1.731,E1 24.8735,E2 232.0036} C_DIS
LIN {X -84.3062,Y -61.9221,Z 108,A -148.2463,B 24.9438,C -1.7325,E1 24.8703,E2 233.9224} C_DIS
LIN {X -86.4172,Y -58.941,Z 108,A -150.031,B 24.9429,C -1.7453,E1 24.8675,E2 235.6852} C_DIS
LIN {X -87.9995,Y -56.5503,Z 108,A -151.8282,B 24.9432,C -1.7412,E1 24.8647,E2 237.5013} C_DIS
LIN {X -89.839,Y -53.5815,Z 108,A -153.6905,B 24.9427,C -1.7481,E1 24.862,E2 239.3567} C_DIS
LIN {X -92.0867,Y -49.6182,Z 108,A -156.3261,B 24.9427,C -1.7498,E1 24.8584,E2 242.002} C_DIS
LIN {X -93.5511,Y -46.7995,Z 108,A -158.1283,B 24.9424,C -1.7524,E1 24.8561,E2 243.8076} C_DIS
LIN {X -95.2102,Y -43.3244,Z 108,A -159.9368,B 24.9413,C -1.7692,E1 24.854,E2 245.5862} C_DIS
LIN {X -96.1355,Y -41.2334,Z 108,A -161.5303,B 24.9419,C -1.7606,E1 24.8522,E2 247.2089} C_DIS
LIN {X -97.4969,Y -37.8991,Z 108,A -163.4791,B 24.9415,C -1.7672,E1 24.8502,E2 249.1528} C_DIS
LIN {X -99.3068,Y -32.8685,Z 108,A -166.2714,B 24.9406,C -1.7807,E1 24.8476,E2 251.9287} C_DIS
LIN {X -100.4042,Y -29.3432,Z 108,A -168.4888,B 24.9406,C -1.78,E1 24.8458,E2 254.1607} C_DIS
LIN {X -101.3394,Y -25.9266,Z 108,A -170.2774,B 24.9399,C -1.7913,E1 24.8446,E2 255.9327} C_DIS
LIN {X -102.1117,Y -22.6986,Z 108,A -172.0859,B 24.9395,C -1.7972,E1 24.8434,E2 257.7376} C_DIS
LIN {X -102.7215,Y -19.752,Z 108,A -173.8428,B 24.9394,C -1.7986,E1 24.8424,E2 259.5018} C_DIS
LIN {X -103.3796,Y -15.9532,Z 108,A -175.9663,B 24.9389,C -1.8048,E1 24.8415,E2 261.6229} C_DIS
LIN {X -103.8576,Y -12.4713,Z 108,A -177.8118,B 24.9383,C -1.8137,E1 24.8408,E2 263.4583} C_DIS
LIN {X -104.1748,Y -9.4592,Z 108,A -179.6413,B 24.9383,C -1.813,E1 24.8403,E2 265.3003} C_DIS
LIN {X -104.4148,Y -6.2991,Z 108,A 178.7921,B 24.9376,C -1.8245,E1 24.84,E2 266.849} C_DIS
LIN {X -104.565,Y -2.8539,Z 108,A 176.7005,B 24.9376,C -1.8235,E1 24.8398,E2 268.9557} C_DIS
LIN {X -104.5988,Y 1.0323,Z 108,A 174.5607,B 24.9372,C -1.83,E1 24.8398,E2 271.0928} C_DIS
LIN {X -104.5389,Y 3.7037,Z 108,A 173.2617,B 24.9365,C -1.8405,E1 24.8399,E2 272.3746} C_DIS
LIN {X -104.4064,Y 6.4443,Z 108,A 171.507,B 24.9368,C -1.8365,E1 24.8402,E2 274.1494} C_DIS
LIN {X -104.0928,Y 10.3369,Z 108,A 169.5899,B 24.9358,C -1.8512,E1 24.8407,E2 276.0429} C_DIS
LIN {X -103.7359,Y 13.4432,Z 108,A 167.8695,B 24.9354,C -1.8565,E1 24.8412,E2 277.761} C_DIS
LIN {X -103.3329,Y 16.2551,Z 108,A 166.2364,B 24.9352,C -1.8588,E1 24.8419,E2 279.3984} C_DIS
LIN {X -102.5978,Y 20.3947,Z 108,A 163.8038,B 24.935,C -1.8616,E1 24.8432,E2 281.8386} C_DIS
LIN {X -101.8801,Y 23.7134,Z 108,A 162.0476,B 24.9344,C -1.8712,E1 24.8442,E2 283.5822} C_DIS
LIN {X -100.9773,Y 27.3026,Z 108,A 160.2374,B 24.9334,C -1.8853,E1 24.8455,E2 285.3694} C_DIS
LIN {X -100.1295,Y 30.269,Z 108,A 158.1729,B 24.9339,C -1.8774,E1 24.8471,E2 287.4646} C_DIS
LIN {X -99.0807,Y 33.5391,Z 108,A 156.4274,B 24.9332,C -1.8881,E1 24.8486,E2 289.1946} C_DIS
LIN {X -97.9095,Y 36.8189,Z 108,A 154.394,B 24.9331,C -1.8896,E1 24.8506,E2 291.2359} C_DIS
LIN {X -96.5278,Y 40.3033,Z 108,A 152.3705,B 24.9325,C -1.8969,E1 24.8527,E2 293.2532} C_DIS
LIN {X -94.9596,Y 43.8703,Z 108,A 149.9133,B 24.9329,C -1.892,E1 24.8556,E2 295.7356} C_DIS
LIN {X -91.8665,Y 50.0243,Z 108,A 146.4554,B 24.9313,C -1.9143,E1 24.86,E2 299.1589} C_DIS
LIN {X -89.7772,Y 53.6859,Z 108,A 144.0364,B 24.9311,C -1.9171,E1 24.8634,E2 301.5838} C_DIS
LIN {X -88.2498,Y 56.1604,Z 108,A 142.4813,B 24.9307,C -1.9229,E1 24.8657,E2 303.1328} C_DIS
LIN {X -86.3468,Y 59.0449,Z 108,A 140.5805,B 24.9303,C -1.9279,E1 24.8686,E2 305.0312} C_DIS
LIN {X -84.6448,Y 61.4596,Z 108,A 139.1687,B 24.9295,C -1.9397,E1 24.8709,E2 306.4218} C_DIS
LIN {X -83.2469,Y 63.342,Z 108,A 137.6046,B 24.9299,C -1.9332,E1 24.8735,E2 308.009} C_DIS
LIN {X -80.8676,Y 66.3527,Z 108,A 135.4312,B 24.9297,C -1.9362,E1 24.8774,E2 310.1853} C_DIS
LIN {X -78.5349,Y 69.096,Z 108,A 133.6065,B 24.929,C -1.9466,E1 24.8807,E2 311.9936} C_DIS
LIN {X -76.2158,Y 71.645,Z 108,A 131.6794,B 24.9287,C -1.9499,E1 24.8843,E2 313.9212} C_DIS
LIN {X -73.5111,Y 74.4175,Z 108,A 129.5615,B 24.9283,C -1.9552,E1 24.8885,E2 316.0356} C_DIS
LIN {X -70.8735,Y 76.934,Z 108,A 127.5183,B 24.9281,C -1.9582,E1 24.8926,E2 318.0798} C_DIS
LIN {X -68.0263,Y 79.4628,Z 108,A 125.4678,B 24.9277,C -1.9642,E1 24.8969,E2 320.1241} C_DIS
LIN {X -65.3473,Y 81.6821,Z 108,A 123.4131,B 24.9277,C -1.963,E1 24.9014,E2 322.1895} C_DIS
LIN {X -62.1992,Y 84.1031,Z 108,A 121.2383,B 24.9274,C -1.9676,E1 24.9062,E2 324.3612} C_DIS
LIN {X -58.8388,Y 86.4864,Z 108,A 119.0966,B 24.9268,C -1.9763,E1 24.9111,E2 326.4894} C_DIS
LIN {X -56.0095,Y 88.3466,Z 108,A 117.1305,B 24.9268,C -1.9758,E1 24.9157,E2 328.4631} C_DIS
LIN {X -52.9662,Y 90.2027,Z 108,A 115.1658,B 24.9266,C -1.9789,E1 24.9205,E2 330.4263} C_DIS
LIN {X -49.9217,Y 91.9221,Z 108,A 113.3705,B 24.926,C -1.9866,E1 24.9248,E2 332.2084} C_DIS
LIN {X -45.7166,Y 94.0853,Z 108,A 110.8187,B 24.9256,C -1.9923,E1 24.9312,E2 334.7538} C_DIS
LIN {X -43.1662,Y 95.2816,Z 108,A 109.3787,B 24.9251,C -1.9984,E1 24.9348,E2 336.1826} C_DIS
LIN {X -40.5616,Y 96.4189,Z 108,A 107.6796,B 24.9253,C -1.9955,E1 24.9392,E2 337.8928} C_DIS
LIN {X -37.4557,Y 97.6684,Z 108,A 105.7537,B 24.9254,C -1.9945,E1 24.9442,E2 339.825} C_DIS
LIN {X -32.3821,Y 99.465,Z 108,A 102.8977,B 24.9249,C -2.0016,E1 24.9517,E2 342.6697} C_DIS
LIN {X -29.4445,Y 100.3742,Z 108,A 101.2941,B 24.9245,C -2.0065,E1 24.9559,E2 344.2644} C_DIS
LIN {X -26.4747,Y 101.1985,Z 108,A 99.6,B 24.9244,C -2.008,E1 24.9605,E2 345.9575} C_DIS
LIN {X -24.1444,Y 101.7805,Z 108,A 98.072,B 24.9249,C -2.0013,E1 24.9647,E2 347.5035} C_DIS
LIN {X -21.238,Y 102.4248,Z 108,A 96.4788,B 24.9247,C -2.0042,E1 24.969,E2 349.0919} C_DIS
LIN {X -17.2994,Y 103.1629,Z 108,A 94.2921,B 24.9245,C -2.0061,E1 24.975,E2 351.2761} C_DIS
LIN {X -13.2651,Y 103.7589,Z 108,A 92.1214,B 24.9243,C -2.0099,E1 24.981,E2 353.4395} C_DIS
LIN {X -9.8009,Y 104.1433,Z 108,A 90.1476,B 24.9243,C -2.0085,E1 24.9865,E2 355.4178} C_DIS
LIN {X -6.2585,Y 104.417,Z 108,A 87.8864,B 24.9252,C -1.9974,E1 24.9929,E2 357.7063} C_DIS
LIN {X -1.5901,Y 104.5917,Z 108,A 85.6018,B 24.9244,C -2.0085,E1 24.9992,E2 359.9648} C_DIS
LIN {X 2.3338,Y 104.578,Z 108,A 83.6698,B 24.9237,C -2.0171,E1 25.0045,E2 361.876} C_DIS
LIN {X 5.1059,Y 104.4804,Z 108,A 81.9025,B 24.9244,C -2.0077,E1 25.0095,E2 363.6652} C_DIS
LIN {X 7.7991,Y 104.3135,Z 108,A 80.4868,B 24.9242,C -2.0101,E1 25.0135,E2 365.0747} C_DIS
LIN {X 11.1024,Y 104.0126,Z 108,A 78.6201,B 24.9244,C -2.0079,E1 25.0187,E2 366.9452} C_DIS
LIN {X 14.065,Y 103.6553,Z 108,A 77.0728,B 24.9242,C -2.0109,E1 25.0229,E2 368.4843} C_DIS
LIN {X 18.1775,Y 103.0123,Z 108,A 74.8745,B 24.924,C -2.0133,E1 25.029,E2 370.6747} C_DIS
LIN {X 21.3282,Y 102.4063,Z 108,A 72.9289,B 24.9246,C -2.0053,E1 25.0343,E2 372.6371} C_DIS
LIN {X 24.3323,Y 101.735,Z 108,A 71.4219,B 24.9241,C -2.0113,E1 25.0384,E2 374.1276} C_DIS
LIN {X 27.0096,Y 101.0565,Z 108,A 69.7797,B 24.9246,C -2.0053,E1 25.0429,E2 375.7815} C_DIS
LIN {X 30.7493,Y 99.9819,Z 108,A 67.4097,B 24.9254,C -1.9944,E1 25.0493,E2 378.1731} C_DIS
LIN {X 34.4172,Y 98.7793,Z 108,A 65.4248,B 24.9252,C -1.9977,E1 25.0545,E2 380.1464} C_DIS
LIN {X 38.3327,Y 97.3266,Z 108,A 63.3392,B 24.9247,C -2.0034,E1 25.0599,E2 382.2139} C_DIS
LIN {X 41.3833,Y 96.0702,Z 108,A 61.3611,B 24.9254,C -1.9947,E1 25.065,E2 384.208} C_DIS
LIN {X 45.1851,Y 94.3407,Z 108,A 59.1729,B 24.9254,C -1.996,E1 25.0705,E2 386.3876} C_DIS
LIN {X 48.1748,Y 92.8518,Z 108,A 57.3072,B 24.9256,C -1.9921,E1 25.0752,E2 388.2573} C_DIS
LIN {X 52.5785,Y 90.4303,Z 108,A 54.5583,B 24.9259,C -1.9884,E1 25.0819,E2 391.0068} C_DIS
LIN {X 55.8671,Y 88.4364,Z 108,A 52.3653,B 24.9264,C -1.9817,E1 25.0871,E2 393.2087} C_DIS
LIN {X 59.4232,Y 86.0863,Z 108,A 50.1895,B 24.9262,C -1.9843,E1 25.0921,E2 395.3711} C_DIS
LIN {X 62.3001,Y 84.0294,Z 108,A 47.8632,B 24.9276,C -1.9652,E1 25.0974,E2 397.7342} C_DIS
LIN {X 64.8971,Y 82.0379,Z 108,A 46.5093,B 24.9265,C -1.9796,E1 25.1003,E2 399.0491} C_DIS
LIN {X 67.7186,Y 79.7249,Z 108,A 44.5743,B 24.9266,C -1.9784,E1 25.1044,E2 400.9796} C_DIS
LIN {X 70.1195,Y 77.6229,Z 108,A 42.9298,B 24.9266,C -1.9791,E1 25.1079,E2 402.6159} C_DIS
LIN {X 73.0555,Y 74.8676,Z 108,A 40.609,B 24.9273,C -1.9697,E1 25.1126,E2 404.9492} C_DIS
LIN {X 76.6635,Y 71.1683,Z 108,A 37.6707,B 24.928,C -1.9591,E1 25.1183,E2 407.8998} C_DIS
LIN {X 78.9852,Y 68.5804,Z 108,A 35.9425,B 24.9278,C -1.962,E1 25.1215,E2 409.6135} C_DIS
LIN {X 81.6905,Y 65.3367,Z 108,A 33.4437,B 24.9288,C -1.9489,E1 25.1259,E2 412.1317} C_DIS
LIN {X 84.0391,Y 62.2869,Z 108,A 31.5706,B 24.9285,C -1.9534,E1 25.129,E2 413.9852} C_DIS
LIN {X 85.2515,Y 60.614,Z 108,A 29.7185,B 24.9308,C -1.921,E1 25.1321,E2 415.9048} C_DIS
LIN {X 87.6448,Y 57.1014,Z 108,A 27.9139,B 24.9297,C -1.9364,E1 25.1348,E2 417.664} C_DIS
LIN {X 89.469,Y 54.1957,Z 108,A 25.8831,B 24.9305,C -1.9252,E1 25.1378,E2 419.7109} C_DIS
LIN {X 91.8091,Y 50.13,Z 108,A 23.6956,B 24.9299,C -1.934,E1 25.1408,E2 421.8663} C_DIS
LIN {X 93.2214,Y 47.4515,Z 108,A 22.0463,B 24.9302,C -1.9298,E1 25.1429,E2 423.5167} C_DIS
LIN {X 95.7336,Y 42.1555,Z 108,A 18.7694,B 24.931,C -1.9179,E1 25.1468,E2 426.804} C_DIS
LIN {X 97.1062,Y 38.8918,Z 108,A 16.4622,B 24.9325,C -1.8969,E1 25.1492,E2 429.148} C_DIS
LIN {X 98.6946,Y 34.6586,Z 108,A 14.4032,B 24.9318,C -1.907,E1 25.1512,E2 431.1717} C_DIS
LIN {X 99.7633,Y 31.4546,Z 108,A 12.4841,B 24.9324,C -1.8985,E1 25.1528,E2 433.1} C_DIS
LIN {X 100.8271,Y 27.8564,Z 108,A 10.6444,B 24.9322,C -1.9013,E1 25.1542,E2 434.9227} C_DIS
LIN {X 101.6259,Y 24.7793,Z 108,A 8.782,B 24.933,C -1.8908,E1 25.1555,E2 436.7989} C_DIS
LIN {X 102.4448,Y 21.1405,Z 108,A 6.83,B 24.9332,C -1.8883,E1 25.1567,E2 438.7455} C_DIS
LIN {X 103.0862,Y 17.7582,Z 108,A 4.8349,B 24.9339,C -1.8777,E1 25.1577,E2 440.7539} C_DIS
LIN {X 103.6492,Y 14.1091,Z 108,A 2.7582,B 24.9345,C -1.869,E1 25.1585,E2 442.8389} C_DIS
LIN {X 104.0044,Y 11.181,Z 108,A 1.0208,B 24.9352,C -1.8588,E1 25.1591,E2 444.5902} C_DIS
LIN {X 104.3881,Y 6.7149,Z 108,A -2.0952,B 24.9377,C -1.8233,E1 25.1597,E2 447.7712} C_DIS
LIN {X 104.596,Y 1.3573,Z 108,A -4.0183,B 24.9354,C -1.8562,E1 25.1597,E2 449.6054} C_DIS
LIN {X 104.554,Y -3.2095,Z 108,A -6.6776,B 24.9364,C -1.8415,E1 25.1597,E2 452.2837} C_DIS
LIN {X 104.3618,Y -7.104,Z 108,A -8.6909,B 24.9366,C -1.8397,E1 25.1593,E2 454.2891} C_DIS
LIN {X 104.053,Y -10.7172,Z 108,A -10.4124,B 24.9362,C -1.8445,E1 25.1589,E2 455.9892} C_DIS
LIN {X 103.6336,Y -14.2186,Z 108,A -12.6427,B 24.9375,C -1.8255,E1 25.1581,E2 458.251} C_DIS
LIN {X 103.1998,Y -17.0784,Z 108,A -14.3391,B 24.9382,C -1.8157,E1 25.1574,E2 459.9606} C_DIS
LIN {X 102.4546,Y -21.0928,Z 108,A -16.3701,B 24.9382,C -1.8172,E1 25.1563,E2 461.9763} C_DIS
LIN {X 101.6566,Y -24.6535,Z 108,A -18.2793,B 24.9382,C -1.8146,E1 25.1551,E2 463.8806} C_DIS
LIN {X 100.6276,Y -28.5646,Z 108,A -20.5723,B 24.939,C -1.8042,E1 25.1534,E2 466.1847} C_DIS
LIN {X 99.323,Y -32.8205,Z 108,A -23.1711,B 24.94,C -1.7897,E1 25.1512,E2 468.803} C_DIS
LIN {X 97.7525,Y -37.2334,Z 108,A -25.6628,B 24.9403,C -1.7849,E1 25.1488,E2 471.2922} C_DIS
LIN {X 96.3623,Y -40.6961,Z 108,A -27.561,B 24.9403,C -1.7847,E1 25.1468,E2 473.1803} C_DIS
LIN {X 95.4746,Y -42.7379,Z 108,A -29.1945,B 24.9417,C -1.7636,E1 25.1449,E2 474.8547} C_DIS
LIN {X 94.0523,Y -45.7853,Z 108,A -30.6982,B 24.9411,C -1.7722,E1 25.1431,E2 476.33} C_DIS
LIN {X 92.4428,Y -48.9514,Z 108,A -32.6121,B 24.9414,C -1.7678,E1 25.1406,E2 478.2443} C_DIS
LIN {X 90.5052,Y -52.4481,Z 108,A -34.89,B 24.9421,C -1.7577,E1 25.1375,E2 480.5342} C_DIS
LIN {X 88.4863,Y -55.7872,Z 108,A -36.9275,B 24.9422,C -1.7557,E1 25.1345,E2 482.566} C_DIS
LIN {X 86.8006,Y -58.3748,Z 108,A -38.5532,B 24.9424,C -1.7537,E1 25.132,E2 484.1884} C_DIS
LIN {X 84.8676,Y -61.1521,Z 108,A -40.8673,B 24.944,C -1.7294,E1 25.1282,E2 486.5487} C_DIS
LIN {X 82.7185,Y -64.0277,Z 108,A -42.3854,B 24.9431,C -1.7427,E1 25.1256,E2 488.0281} C_DIS
LIN {X 80.4837,Y -66.8148,Z 108,A -44.1485,B 24.9429,C -1.7456,E1 25.1226,E2 489.7762} C_DIS
LIN {X 77.4814,Y -70.2754,Z 108,A -46.8555,B 24.9439,C -1.7309,E1 25.1175,E2 492.5058} C_DIS
LIN {X 73.8313,Y -74.1012,Z 108,A -49.6902,B 24.9442,C -1.7262,E1 25.112,E2 495.3392} C_DIS
LIN {X 69.4144,Y -78.2542,Z 108,A -53.0295,B 24.9447,C -1.7176,E1 25.1052,E2 498.6853} C_DIS
LIN {X 66.7026,Y -80.577,Z 108,A -54.9745,B 24.945,C -1.7136,E1 25.101,E2 500.6322} C_DIS
LIN {X 63.9005,Y -82.8166,Z 108,A -56.6205,B 24.9444,C -1.7225,E1 25.0974,E2 502.2511} C_DIS
Enddeposition()
END
